LIN {X 0,Y 234.996,Z 198.211,A -85,B 0,C 180,E1 -19773.794,E2 -19773.794} C_VEL
LIN {X 0,Y 235.014,Z 198.209,A -85,B 0,C 180,E1 -19778.97,E2 -19778.97} C_VEL
LIN {X 0,Y 235.098,Z 198.197,A -85,B 0,C 180,E1 -19783.059,E2 -19783.059} C_VEL
LIN {X 0,Y 235.115,Z 198.198,A -85,B 0,C 180,E1 -19787.922,E2 -19787.922} C_VEL
LIN {X 0,Y 235.32,Z 198.173,A -85,B 0,C 180,E1 -19791.412,E2 -19791.412} C_VEL
LIN {X 0,Y 235.356,Z 198.167,A -85,B 0,C 180,E1 -19793.14,E2 -19793.14} C_VEL
LIN {X 0,Y 235.595,Z 198.137,A -85,B 0,C 180,E1 -19798.29,E2 -19798.29} C_VEL
LIN {X 0,Y 235.595,Z 198.138,A -85,B 0,C 180,E1 -19801.709,E2 -19801.709} C_VEL
LIN {X 0,Y 235.351,Z 198.171,A -85,B 0,C 180,E1 -19806.86,E2 -19806.86} C_VEL
LIN {X 0,Y 235.216,Z 198.186,A -85,B 0,C 180,E1 -19810.327,E2 -19810.327} C_VEL
LIN {X 0,Y 235.116,Z 198.199,A -85,B 0,C 180,E1 -19815.606,E2 -19815.606} C_VEL
LIN {X 0,Y 235.009,Z 198.212,A -85,B 0,C 180,E1 -19819.206,E2 -19819.206} C_VEL
LIN {X 0,Y 234.954,Z 198.218,A -85,B 0,C 180,E1 -19822.884,E2 -19822.884} C_VEL
LIN {X 0,Y 234.969,Z 198.217,A -85,B 0,C 180,E1 -19826.657,E2 -19826.657} C_VEL
LIN {X 0,Y 234.924,Z 198.224,A -85,B 0,C 180,E1 -19830.569,E2 -19830.569} C_VEL
LIN {X 0,Y 234.927,Z 198.224,A -85,B 0,C 180,E1 -19834.639,E2 -19834.639} C_VEL
LIN {X 0,Y 234.931,Z 198.302,A -85,B 0,C 180,E1 -19837.285,E2 -19837.285} C_VEL
LIN {X 0,Y 235.419,Z 201.2,A -85,B 0,C 180,E1 -19841.054,E2 -19841.054} C_VEL
LIN {X 0,Y 236.071,Z 204.999,A -85,B 0,C 180,E1 -19845.602,E2 -19845.602} C_VEL
LIN {X 0,Y 236.628,Z 208.216,A -85,B 0,C 180,E1 -19849.2,E2 -19849.2} C_VEL
LIN {X 0,Y 236.793,Z 209.756,A -85,B 0,C 180,E1 -19850.844,E2 -19850.844} C_VEL
LIN {X 0,Y 236.138,Z 210.744,A -85,B 0,C 180,E1 -19851.757,E2 -19851.757} C_VEL
LIN {X 0,Y 233.277,Z 212.555,A -85,B 0,C 180,E1 -19853.17,E2 -19853.17} C_VEL
LIN {X 0,Y 230.314,Z 214.382,A -85,B 0,C 180,E1 -19854.615,E2 -19854.615} C_VEL
LIN {X 0,Y 229.548,Z 215.411,A -85,B 0,C 180,E1 -19855.565,E2 -19855.565} C_VEL
LIN {X 0,Y 229.157,Z 217.081,A -85,B 0,C 180,E1 -19857.204,E2 -19857.204} C_VEL
LIN {X 0,Y 230.079,Z 220.478,A -85,B 0,C 180,E1 -19857.555,E2 -19857.555} C_VEL
LIN {X 0,Y 233.635,Z 233.062,A -85,B 0,C 180,E1 -19858.962,E2 -19858.962} C_VEL
LIN {X 0,Y 236.089,Z 245.694,A -85,B 0,C 180,E1 -19860.544,E2 -19860.544} C_VEL
LIN {X 0,Y 237.459,Z 257.416,A -85,B 0,C 180,E1 -19862.24,E2 -19862.24} C_VEL
LIN {X 0,Y 237.895,Z 268.917,A -85,B 0,C 180,E1 -19864.167,E2 -19864.167} C_VEL
LIN {X 0,Y 237.714,Z 273.85,A -85,B 0,C 180,E1 -19865.083,E2 -19865.083} C_VEL
LIN {X 0,Y 235.107,Z 284.313,A -85,B 0,C 180,E1 -19867.132,E2 -19867.132} C_VEL
LIN {X 0,Y 232.903,Z 293.005,A -85,B 0,C 180,E1 -19869.3,E2 -19869.3} C_VEL
LIN {X 0,Y 230.721,Z 301.061,A -85,B 0,C 180,E1 -19871.806,E2 -19871.806} C_VEL
LIN {X 0,Y 228.899,Z 307.733,A -85,B 0,C 180,E1 -19874.415,E2 -19874.415} C_VEL
LIN {X 0,Y 227.307,Z 313.84,A -85,B 0,C 180,E1 -19877.5,E2 -19877.5} C_VEL
LIN {X 0,Y 226.433,Z 317.814,A -85,B 0,C 180,E1 -19880.171,E2 -19880.171} C_VEL
LIN {X 0,Y 225.852,Z 320.751,A -85,B 0,C 180,E1 -19882.849,E2 -19882.849} C_VEL
LIN {X 0,Y 225.617,Z 322.647,A -85,B 0,C 180,E1 -19885.419,E2 -19885.419} C_VEL
LIN {X 0,Y 225.662,Z 323.764,A -85,B 0,C 180,E1 -19888.215,E2 -19888.215} C_VEL
LIN {X 0,Y 225.698,Z 323.979,A -85,B 0,C 180,E1 -19890,E2 -19890} C_VEL
LIN {X 0,Y 225.662,Z 323.756,A -85,B 0,C 180,E1 -19891.784,E2 -19891.784} C_VEL
LIN {X 0,Y 225.69,Z 322.134,A -85,B 0,C 180,E1 -19895.36,E2 -19895.36} C_VEL
LIN {X 0,Y 225.852,Z 320.726,A -85,B 0,C 180,E1 -19897.15,E2 -19897.15} C_VEL
LIN {X 0,Y 226.432,Z 317.777,A -85,B 0,C 180,E1 -19899.829,E2 -19899.829} C_VEL
LIN {X 0,Y 227.306,Z 313.787,A -85,B 0,C 180,E1 -19902.499,E2 -19902.499} C_VEL
LIN {X 0,Y 228.896,Z 307.66,A -85,B 0,C 180,E1 -19905.584,E2 -19905.584} C_VEL
LIN {X 0,Y 230.72,Z 300.972,A -85,B 0,C 180,E1 -19908.193,E2 -19908.193} C_VEL
LIN {X 0,Y 232.846,Z 293.03,A -85,B 0,C 180,E1 -19910.662,E2 -19910.662} C_VEL
LIN {X 0,Y 235.071,Z 284.172,A -85,B 0,C 180,E1 -19912.871,E2 -19912.871} C_VEL
LIN {X 0,Y 237.68,Z 273.673,A -85,B 0,C 180,E1 -19914.92,E2 -19914.92} C_VEL
LIN {X 0,Y 237.822,Z 264.985,A -85,B 0,C 180,E1 -19916.493,E2 -19916.493} C_VEL
LIN {X 0,Y 237.081,Z 253.496,A -85,B 0,C 180,E1 -19918.313,E2 -19918.313} C_VEL
LIN {X 0,Y 235.519,Z 242.287,A -85,B 0,C 180,E1 -19919.86,E2 -19919.86} C_VEL
LIN {X 0,Y 232.684,Z 229.401,A -85,B 0,C 180,E1 -19921.431,E2 -19921.431} C_VEL
LIN {X 0,Y 229.162,Z 217.507,A -85,B 0,C 180,E1 -19922.7,E2 -19922.7} C_VEL
LIN {X 0,Y 229.124,Z 217.065,A -85,B 0,C 180,E1 -19922.774,E2 -19922.774} C_VEL
LIN {X 0,Y 229.714,Z 214.269,A -85,B 0,C 180,E1 -19925.541,E2 -19925.541} C_VEL
LIN {X 0,Y 229.838,Z 211.122,A -85,B 0,C 180,E1 -19928.817,E2 -19928.817} C_VEL
LIN {X 0,Y 229.356,Z 207.677,A -85,B 0,C 180,E1 -19932.658,E2 -19932.658} C_VEL
LIN {X 0,Y 228.641,Z 203.611,A -85,B 0,C 180,E1 -19937.536,E2 -19937.536} C_VEL
LIN {X 0,Y 228.102,Z 200.24,A -85,B 0,C 180,E1 -19941.96,E2 -19941.96} C_VEL
LIN {X 0,Y 227.872,Z 199.103,A -85,B 0,C 180,E1 -19943.708,E2 -19943.708} C_VEL
LIN {X 0,Y 227.865,Z 199.102,A -85,B 0,C 180,E1 -19948.377,E2 -19948.377} C_VEL
LIN {X 0,Y 227.877,Z 199.101,A -85,B 0,C 180,E1 -19952.444,E2 -19952.444} C_VEL
LIN {X 0,Y 227.905,Z 199.099,A -85,B 0,C 180,E1 -19956.366,E2 -19956.366} C_VEL
LIN {X 0,Y 227.936,Z 199.094,A -85,B 0,C 180,E1 -19960.174,E2 -19960.174} C_VEL
LIN {X 0,Y 228.056,Z 199.078,A -85,B 0,C 180,E1 -19963.898,E2 -19963.898} C_VEL
LIN {X 0,Y 228.07,Z 199.075,A -85,B 0,C 180,E1 -19967.543,E2 -19967.543} C_VEL
LIN {X 0,Y 228.251,Z 199.053,A -85,B 0,C 180,E1 -19971.144,E2 -19971.144} C_VEL
LIN {X 0,Y 228.3,Z 199.047,A -85,B 0,C 180,E1 -19972.927,E2 -19972.927} C_VEL
LIN {X 0,Y 228.55,Z 199.014,A -85,B 0,C 180,E1 -19978.238,E2 -19978.238} C_VEL
LIN {X 0,Y 228.55,Z 199.014,A -85,B 0,C 180,E1 -19981.762,E2 -19981.762} C_VEL
LIN {X 0,Y 228.305,Z 199.045,A -85,B 0,C 180,E1 -19987.073,E2 -19987.073} C_VEL
LIN {X 0,Y 228.144,Z 199.067,A -85,B 0,C 180,E1 -19990.651,E2 -19990.651} C_VEL
LIN {X 0,Y 228.063,Z 199.078,A -85,B 0,C 180,E1 -19994.272,E2 -19994.272} C_VEL
LIN {X 0,Y 228.002,Z 199.084,A -85,B 0,C 180,E1 -19997.954,E2 -19997.954} C_VEL
LIN {X 0,Y 227.929,Z 199.093,A -85,B 0,C 180,E1 -20002.33,E2 -20002.33} C_VEL
LIN {X 0,Y 227.942,Z 199.091,A -85,B 0,C 180,E1 -20006.603,E2 -20006.603} C_VEL
LIN {X 0,Y 227.907,Z 199.096,A -85,B 0,C 180,E1 -20010.296,E2 -20010.296} C_VEL
LIN {X 0,Y 227.875,Z 199.102,A -85,B 0,C 180,E1 -20013.721,E2 -20013.721} C_VEL
LIN {X 0,Y 227.839,Z 199.106,A -85,B 0,C 180,E1 -20018.092,E2 -20018.092} C_VEL
LIN {X 0,Y 227.805,Z 199.11,A -85,B 0,C 180,E1 -20022.744,E2 -20022.744} C_VEL
LIN {X 0,Y 227.825,Z 199.107,A -85,B 0,C 180,E1 -20025.195,E2 -20025.195} C_VEL
LIN {X 0,Y 227.904,Z 199.685,A -85,B 0,C 180,E1 -20027.74,E2 -20027.74} C_VEL
LIN {X 0,Y 228.203,Z 202.454,A -85,B 0,C 180,E1 -20031.98,E2 -20031.98} C_VEL
LIN {X 0,Y 228.228,Z 204.017,A -85,B 0,C 180,E1 -20034.192,E2 -20034.192} C_VEL
LIN {X 0,Y 228.051,Z 206.435,A -85,B 0,C 180,E1 -20037.19,E2 -20037.19} C_VEL
LIN {X 0,Y 229.183,Z 209.556,A -85,B 0,C 180,E1 -20037.548,E2 -20037.548} C_VEL
LIN {X 0,Y 233.35,Z 220.919,A -85,B 0,C 180,E1 -20039.001,E2 -20039.001} C_VEL
LIN {X 0,Y 236.465,Z 231.896,A -85,B 0,C 180,E1 -20040.528,E2 -20040.528} C_VEL
LIN {X 0,Y 238.564,Z 242.208,A -85,B 0,C 180,E1 -20042.103,E2 -20042.103} C_VEL
LIN {X 0,Y 239.656,Z 251.285,A -85,B 0,C 180,E1 -20043.631,E2 -20043.631} C_VEL
LIN {X 0,Y 239.798,Z 255.538,A -85,B 0,C 180,E1 -20044.387,E2 -20044.387} C_VEL
LIN {X 0,Y 237.438,Z 265.983,A -85,B 0,C 180,E1 -20046.217,E2 -20046.217} C_VEL
LIN {X 0,Y 235.445,Z 274.952,A -85,B 0,C 180,E1 -20048.209,E2 -20048.209} C_VEL
LIN {X 0,Y 233.002,Z 283.746,A -85,B 0,C 180,E1 -20050.623,E2 -20050.623} C_VEL
LIN {X 0,Y 230.82,Z 291.15,A -85,B 0,C 180,E1 -20053.187,E2 -20053.187} C_VEL
LIN {X 0,Y 229.103,Z 297.087,A -85,B 0,C 180,E1 -20055.794,E2 -20055.794} C_VEL
LIN {X 0,Y 227.751,Z 301.777,A -85,B 0,C 180,E1 -20058.43,E2 -20058.43} C_VEL
LIN {X 0,Y 226.85,Z 305.362,A -85,B 0,C 180,E1 -20061.089,E2 -20061.089} C_VEL
LIN {X 0,Y 226.238,Z 307.944,A -85,B 0,C 180,E1 -20063.759,E2 -20063.759} C_VEL
LIN {X 0,Y 225.888,Z 309.593,A -85,B 0,C 180,E1 -20066.433,E2 -20066.433} C_VEL
LIN {X 0,Y 225.781,Z 310.2,A -85,B 0,C 180,E1 -20068.217,E2 -20068.217} C_VEL
LIN {X 0,Y 225.751,Z 310.428,A -85,B 0,C 180,E1 -20070,E2 -20070} C_VEL
LIN {X 0,Y 225.781,Z 310.234,A -85,B 0,C 180,E1 -20071.784,E2 -20071.784} C_VEL
LIN {X 0,Y 225.886,Z 309.648,A -85,B 0,C 180,E1 -20073.568,E2 -20073.568} C_VEL
LIN {X 0,Y 226.395,Z 307.325,A -85,B 0,C 180,E1 -20077.133,E2 -20077.133} C_VEL
LIN {X 0,Y 227.097,Z 304.458,A -85,B 0,C 180,E1 -20079.8,E2 -20079.8} C_VEL
LIN {X 0,Y 228.133,Z 300.57,A -85,B 0,C 180,E1 -20082.454,E2 -20082.454} C_VEL
LIN {X 0,Y 229.598,Z 295.549,A -85,B 0,C 180,E1 -20085.081,E2 -20085.081} C_VEL
LIN {X 0,Y 231.424,Z 289.226,A -85,B 0,C 180,E1 -20087.679,E2 -20087.679} C_VEL
LIN {X 0,Y 233.778,Z 281.307,A -85,B 0,C 180,E1 -20090.226,E2 -20090.226} C_VEL
LIN {X 0,Y 235.841,Z 273.317,A -85,B 0,C 180,E1 -20092.311,E2 -20092.311} C_VEL
LIN {X 0,Y 238.119,Z 263.394,A -85,B 0,C 180,E1 -20094.407,E2 -20094.407} C_VEL
LIN {X 0,Y 239.946,Z 254.985,A -85,B 0,C 180,E1 -20095.829,E2 -20095.829} C_VEL
LIN {X 0,Y 239.038,Z 245.57,A -85,B 0,C 180,E1 -20097.485,E2 -20097.485} C_VEL
LIN {X 0,Y 237.134,Z 234.687,A -85,B 0,C 180,E1 -20099.199,E2 -20099.199} C_VEL
LIN {X 0,Y 234.237,Z 223.714,A -85,B 0,C 180,E1 -20100.768,E2 -20100.768} C_VEL
LIN {X 0,Y 230.381,Z 212.541,A -85,B 0,C 180,E1 -20102.23,E2 -20102.23} C_VEL
LIN {X 0,Y 228.147,Z 206.8,A -85,B 0,C 180,E1 -20102.921,E2 -20102.921} C_VEL
LIN {X 0,Y 228.042,Z 206.204,A -85,B 0,C 180,E1 -20103.008,E2 -20103.008} C_VEL
LIN {X 0,Y 228.249,Z 203.403,A -85,B 0,C 180,E1 -20106.816,E2 -20106.816} C_VEL
LIN {X 0,Y 228.079,Z 201.029,A -85,B 0,C 180,E1 -20110.323,E2 -20110.323} C_VEL
LIN {X 0,Y 227.866,Z 199.496,A -85,B 0,C 180,E1 -20112.73,E2 -20112.73} C_VEL
LIN {X 0,Y 227.824,Z 199.105,A -85,B 0,C 180,E1 -20115.196,E2 -20115.196} C_VEL
LIN {X 0,Y 227.827,Z 199.107,A -85,B 0,C 180,E1 -20119.623,E2 -20119.623} C_VEL
LIN {X 0,Y 227.867,Z 199.102,A -85,B 0,C 180,E1 -20124.125,E2 -20124.125} C_VEL
LIN {X 0,Y 227.868,Z 199.1,A -85,B 0,C 180,E1 -20128.377,E2 -20128.377} C_VEL
LIN {X 0,Y 227.881,Z 199.1,A -85,B 0,C 180,E1 -20132.444,E2 -20132.444} C_VEL
LIN {X 0,Y 227.916,Z 199.095,A -85,B 0,C 180,E1 -20136.367,E2 -20136.367} C_VEL
LIN {X 0,Y 227.945,Z 199.092,A -85,B 0,C 180,E1 -20140.175,E2 -20140.175} C_VEL
LIN {X 0,Y 228.06,Z 199.078,A -85,B 0,C 180,E1 -20143.898,E2 -20143.898} C_VEL
LIN {X 0,Y 228.074,Z 199.076,A -85,B 0,C 180,E1 -20147.543,E2 -20147.543} C_VEL
LIN {X 0,Y 228.259,Z 199.051,A -85,B 0,C 180,E1 -20151.144,E2 -20151.144} C_VEL
LIN {X 0,Y 228.308,Z 199.045,A -85,B 0,C 180,E1 -20152.927,E2 -20152.927} C_VEL
LIN {X 0,Y 228.553,Z 199.014,A -85,B 0,C 180,E1 -20158.238,E2 -20158.238} C_VEL
LIN {X 0,Y 228.554,Z 199.015,A -85,B 0,C 180,E1 -20161.762,E2 -20161.762} C_VEL
LIN {X 0,Y 228.303,Z 199.048,A -85,B 0,C 180,E1 -20167.073,E2 -20167.073} C_VEL
LIN {X 0,Y 228.148,Z 199.069,A -85,B 0,C 180,E1 -20170.651,E2 -20170.651} C_VEL
LIN {X 0,Y 228.067,Z 199.078,A -85,B 0,C 180,E1 -20174.272,E2 -20174.272} C_VEL
LIN {X 0,Y 228.005,Z 199.086,A -85,B 0,C 180,E1 -20177.953,E2 -20177.953} C_VEL
LIN {X 0,Y 227.918,Z 199.095,A -85,B 0,C 180,E1 -20182.321,E2 -20182.321} C_VEL
LIN {X 0,Y 227.943,Z 199.093,A -85,B 0,C 180,E1 -20186.602,E2 -20186.602} C_VEL
LIN {X 0,Y 227.898,Z 199.1,A -85,B 0,C 180,E1 -20190.291,E2 -20190.291} C_VEL
LIN {X 0,Y 227.878,Z 199.104,A -85,B 0,C 180,E1 -20193.72,E2 -20193.72} C_VEL
LIN {X 0,Y 227.898,Z 199.226,A -85,B 0,C 180,E1 -20196.536,E2 -20196.536} C_VEL
LIN {X 0,Y 228.347,Z 201.962,A -85,B 0,C 180,E1 -20200.266,E2 -20200.266} C_VEL
LIN {X 0,Y 228.97,Z 205.655,A -85,B 0,C 180,E1 -20204.907,E2 -20204.907} C_VEL
LIN {X 0,Y 229.573,Z 209.041,A -85,B 0,C 180,E1 -20208.839,E2 -20208.839} C_VEL
LIN {X 0,Y 229.805,Z 212.223,A -85,B 0,C 180,E1 -20212.291,E2 -20212.291} C_VEL
LIN {X 0,Y 229.548,Z 215.411,A -85,B 0,C 180,E1 -20215.565,E2 -20215.565} C_VEL
LIN {X 0,Y 229.593,Z 217.095,A -85,B 0,C 180,E1 -20216.397,E2 -20216.397} C_VEL
LIN {X 0,Y 229.787,Z 219.822,A -85,B 0,C 180,E1 -20217.055,E2 -20217.055} C_VEL
LIN {X 0,Y 229.991,Z 225.007,A -85,B 0,C 180,E1 -20217.764,E2 -20217.764} C_VEL
LIN {X 0,Y 229.616,Z 235.258,A -85,B 0,C 180,E1 -20218.556,E2 -20218.556} C_VEL
LIN {X 0,Y 228.975,Z 241.389,A -85,B 0,C 180,E1 -20219.076,E2 -20219.076} C_VEL
LIN {X 0,Y 229.077,Z 243.326,A -85,B 0,C 180,E1 -20219.308,E2 -20219.308} C_VEL
LIN {X 0,Y 230.659,Z 255.124,A -85,B 0,C 180,E1 -20221.043,E2 -20221.043} C_VEL
LIN {X 0,Y 231.247,Z 266.076,A -85,B 0,C 180,E1 -20222.878,E2 -20222.878} C_VEL
LIN {X 0,Y 231.01,Z 274.817,A -85,B 0,C 180,E1 -20224.55,E2 -20224.55} C_VEL
LIN {X 0,Y 228.563,Z 284.102,A -85,B 0,C 180,E1 -20226.438,E2 -20226.438} C_VEL
LIN {X 0,Y 226.032,Z 293.522,A -85,B 0,C 180,E1 -20228.874,E2 -20228.874} C_VEL
LIN {X 0,Y 223.962,Z 300.849,A -85,B 0,C 180,E1 -20231.237,E2 -20231.237} C_VEL
LIN {X 0,Y 222.046,Z 307.521,A -85,B 0,C 180,E1 -20233.922,E2 -20233.922} C_VEL
LIN {X 0,Y 220.351,Z 313.627,A -85,B 0,C 180,E1 -20237.099,E2 -20237.099} C_VEL
LIN {X 0,Y 219.405,Z 317.601,A -85,B 0,C 180,E1 -20239.852,E2 -20239.852} C_VEL
LIN {X 0,Y 218.803,Z 320.538,A -85,B 0,C 180,E1 -20242.618,E2 -20242.618} C_VEL
LIN {X 0,Y 218.52,Z 322.61,A -85,B 0,C 180,E1 -20245.574,E2 -20245.574} C_VEL
LIN {X 0,Y 218.56,Z 323.551,A -85,B 0,C 180,E1 -20248.157,E2 -20248.157} C_VEL
LIN {X 0,Y 218.614,Z 323.766,A -85,B 0,C 180,E1 -20250,E2 -20250} C_VEL
LIN {X 0,Y 218.56,Z 323.542,A -85,B 0,C 180,E1 -20251.842,E2 -20251.842} C_VEL
LIN {X 0,Y 218.554,Z 322.534,A -85,B 0,C 180,E1 -20254.538,E2 -20254.538} C_VEL
LIN {X 0,Y 218.803,Z 320.512,A -85,B 0,C 180,E1 -20257.381,E2 -20257.381} C_VEL
LIN {X 0,Y 219.404,Z 317.562,A -85,B 0,C 180,E1 -20260.147,E2 -20260.147} C_VEL
LIN {X 0,Y 220.35,Z 313.572,A -85,B 0,C 180,E1 -20262.9,E2 -20262.9} C_VEL
LIN {X 0,Y 222.044,Z 307.444,A -85,B 0,C 180,E1 -20266.078,E2 -20266.078} C_VEL
LIN {X 0,Y 223.96,Z 300.756,A -85,B 0,C 180,E1 -20268.762,E2 -20268.762} C_VEL
LIN {X 0,Y 225.999,Z 293.482,A -85,B 0,C 180,E1 -20271.104,E2 -20271.104} C_VEL
LIN {X 0,Y 228.517,Z 283.955,A -85,B 0,C 180,E1 -20273.566,E2 -20273.566} C_VEL
LIN {X 0,Y 231.127,Z 273.451,A -85,B 0,C 180,E1 -20275.677,E2 -20275.677} C_VEL
LIN {X 0,Y 231.116,Z 262.504,A -85,B 0,C 180,E1 -20277.709,E2 -20277.709} C_VEL
LIN {X 0,Y 230.318,Z 251.884,A -85,B 0,C 180,E1 -20279.417,E2 -20279.417} C_VEL
LIN {X 0,Y 228.386,Z 239.706,A -85,B 0,C 180,E1 -20281.145,E2 -20281.145} C_VEL
LIN {X 0,Y 225.462,Z 227.374,A -85,B 0,C 180,E1 -20282.687,E2 -20282.687} C_VEL
LIN {X 0,Y 222.418,Z 217.479,A -85,B 0,C 180,E1 -20283.812,E2 -20283.812} C_VEL
LIN {X 0,Y 222.355,Z 216.881,A -85,B 0,C 180,E1 -20283.862,E2 -20283.862} C_VEL
LIN {X 0,Y 222.793,Z 213,A -85,B 0,C 180,E1 -20287.943,E2 -20287.943} C_VEL
LIN {X 0,Y 222.632,Z 210.496,A -85,B 0,C 180,E1 -20290.744,E2 -20290.744} C_VEL
LIN {X 0,Y 222.122,Z 207.666,A -85,B 0,C 180,E1 -20294.113,E2 -20294.113} C_VEL
LIN {X 0,Y 221.554,Z 204.406,A -85,B 0,C 180,E1 -20298.229,E2 -20298.229} C_VEL
LIN {X 0,Y 221.028,Z 201.065,A -85,B 0,C 180,E1 -20302.833,E2 -20302.833} C_VEL
LIN {X 0,Y 220.812,Z 199.981,A -85,B 0,C 180,E1 -20304.489,E2 -20304.489} C_VEL
LIN {X 0,Y 220.832,Z 199.977,A -85,B 0,C 180,E1 -20309.389,E2 -20309.389} C_VEL
LIN {X 0,Y 220.892,Z 199.972,A -85,B 0,C 180,E1 -20313.549,E2 -20313.549} C_VEL
LIN {X 0,Y 220.864,Z 199.976,A -85,B 0,C 180,E1 -20317.552,E2 -20317.552} C_VEL
LIN {X 0,Y 220.983,Z 199.959,A -85,B 0,C 180,E1 -20322.571,E2 -20322.571} C_VEL
LIN {X 0,Y 221.01,Z 199.956,A -85,B 0,C 180,E1 -20327.138,E2 -20327.138} C_VEL
LIN {X 0,Y 221.192,Z 199.931,A -85,B 0,C 180,E1 -20330.859,E2 -20330.859} C_VEL
LIN {X 0,Y 221.122,Z 199.941,A -85,B 0,C 180,E1 -20334.529,E2 -20334.529} C_VEL
LIN {X 0,Y 221.508,Z 199.891,A -85,B 0,C 180,E1 -20338.182,E2 -20338.182} C_VEL
LIN {X 0,Y 221.508,Z 199.891,A -85,B 0,C 180,E1 -20341.818,E2 -20341.818} C_VEL
LIN {X 0,Y 221.243,Z 199.924,A -85,B 0,C 180,E1 -20347.3,E2 -20347.3} C_VEL
LIN {X 0,Y 221.066,Z 199.948,A -85,B 0,C 180,E1 -20350.997,E2 -20350.997} C_VEL
LIN {X 0,Y 220.994,Z 199.956,A -85,B 0,C 180,E1 -20354.739,E2 -20354.739} C_VEL
LIN {X 0,Y 220.921,Z 199.966,A -85,B 0,C 180,E1 -20358.55,E2 -20358.55} C_VEL
LIN {X 0,Y 220.895,Z 199.968,A -85,B 0,C 180,E1 -20362.683,E2 -20362.683} C_VEL
LIN {X 0,Y 220.885,Z 199.971,A -85,B 0,C 180,E1 -20367.016,E2 -20367.016} C_VEL
LIN {X 0,Y 220.837,Z 199.976,A -85,B 0,C 180,E1 -20370.768,E2 -20370.768} C_VEL
LIN {X 0,Y 220.792,Z 199.983,A -85,B 0,C 180,E1 -20374.957,E2 -20374.957} C_VEL
LIN {X 0,Y 220.8,Z 199.98,A -85,B 0,C 180,E1 -20377.276,E2 -20377.276} C_VEL
LIN {X 0,Y 220.794,Z 199.982,A -85,B 0,C 180,E1 -20380.189,E2 -20380.189} C_VEL
LIN {X 0,Y 220.767,Z 199.986,A -85,B 0,C 180,E1 -20384.456,E2 -20384.456} C_VEL
LIN {X 0,Y 220.776,Z 199.984,A -85,B 0,C 180,E1 -20385.547,E2 -20385.547} C_VEL
LIN {X 0,Y 220.949,Z 201.161,A -85,B 0,C 180,E1 -20388.09,E2 -20388.09} C_VEL
LIN {X 0,Y 221.149,Z 202.697,A -85,B 0,C 180,E1 -20390.537,E2 -20390.537} C_VEL
LIN {X 0,Y 221.222,Z 204.251,A -85,B 0,C 180,E1 -20392.872,E2 -20392.872} C_VEL
LIN {X 0,Y 221.073,Z 206.476,A -85,B 0,C 180,E1 -20396.005,E2 -20396.005} C_VEL
LIN {X 0,Y 222.205,Z 209.663,A -85,B 0,C 180,E1 -20396.386,E2 -20396.386} C_VEL
LIN {X 0,Y 226.427,Z 220.676,A -85,B 0,C 180,E1 -20397.899,E2 -20397.899} C_VEL
LIN {X 0,Y 229.58,Z 231.463,A -85,B 0,C 180,E1 -20399.474,E2 -20399.474} C_VEL
LIN {X 0,Y 231.954,Z 242.834,A -85,B 0,C 180,E1 -20401.291,E2 -20401.291} C_VEL
LIN {X 0,Y 233.148,Z 253.158,A -85,B 0,C 180,E1 -20403.118,E2 -20403.118} C_VEL
LIN {X 0,Y 233.139,Z 257.042,A -85,B 0,C 180,E1 -20403.841,E2 -20403.841} C_VEL
LIN {X 0,Y 230.721,Z 267.252,A -85,B 0,C 180,E1 -20405.719,E2 -20405.719} C_VEL
LIN {X 0,Y 228.477,Z 276.713,A -85,B 0,C 180,E1 -20407.955,E2 -20407.955} C_VEL
LIN {X 0,Y 225.927,Z 285.309,A -85,B 0,C 180,E1 -20410.464,E2 -20410.464} C_VEL
LIN {X 0,Y 223.73,Z 292.473,A -85,B 0,C 180,E1 -20413.109,E2 -20413.109} C_VEL
LIN {X 0,Y 222.221,Z 297.302,A -85,B 0,C 180,E1 -20415.345,E2 -20415.345} C_VEL
LIN {X 0,Y 220.806,Z 301.992,A -85,B 0,C 180,E1 -20418.06,E2 -20418.06} C_VEL
LIN {X 0,Y 219.831,Z 305.576,A -85,B 0,C 180,E1 -20420.802,E2 -20420.802} C_VEL
LIN {X 0,Y 219.119,Z 308.408,A -85,B 0,C 180,E1 -20423.878,E2 -20423.878} C_VEL
LIN {X 0,Y 218.8,Z 309.806,A -85,B 0,C 180,E1 -20426.317,E2 -20426.317} C_VEL
LIN {X 0,Y 218.7,Z 310.413,A -85,B 0,C 180,E1 -20428.159,E2 -20428.159} C_VEL
LIN {X 0,Y 218.666,Z 310.641,A -85,B 0,C 180,E1 -20430,E2 -20430} C_VEL
LIN {X 0,Y 218.699,Z 310.447,A -85,B 0,C 180,E1 -20431.842,E2 -20431.842} C_VEL
LIN {X 0,Y 219.015,Z 308.894,A -85,B 0,C 180,E1 -20435.525,E2 -20435.525} C_VEL
LIN {X 0,Y 219.352,Z 307.537,A -85,B 0,C 180,E1 -20437.364,E2 -20437.364} C_VEL
LIN {X 0,Y 220.097,Z 304.671,A -85,B 0,C 180,E1 -20440.115,E2 -20440.115} C_VEL
LIN {X 0,Y 221.208,Z 300.781,A -85,B 0,C 180,E1 -20442.85,E2 -20442.85} C_VEL
LIN {X 0,Y 222.754,Z 295.761,A -85,B 0,C 180,E1 -20445.556,E2 -20445.556} C_VEL
LIN {X 0,Y 224.669,Z 289.437,A -85,B 0,C 180,E1 -20448.229,E2 -20448.229} C_VEL
LIN {X 0,Y 227.143,Z 281.517,A -85,B 0,C 180,E1 -20450.844,E2 -20450.844} C_VEL
LIN {X 0,Y 229.155,Z 274.045,A -85,B 0,C 180,E1 -20452.859,E2 -20452.859} C_VEL
LIN {X 0,Y 231.392,Z 264.669,A -85,B 0,C 180,E1 -20454.925,E2 -20454.925} C_VEL
LIN {X 0,Y 233.283,Z 256.481,A -85,B 0,C 180,E1 -20456.383,E2 -20456.383} C_VEL
LIN {X 0,Y 232.765,Z 248.766,A -85,B 0,C 180,E1 -20457.823,E2 -20457.823} C_VEL
LIN {X 0,Y 231.143,Z 238.24,A -85,B 0,C 180,E1 -20459.606,E2 -20459.606} C_VEL
LIN {X 0,Y 228.364,Z 226.928,A -85,B 0,C 180,E1 -20461.348,E2 -20461.348} C_VEL
LIN {X 0,Y 224.773,Z 216.012,A -85,B 0,C 180,E1 -20462.897,E2 -20462.897} C_VEL
LIN {X 0,Y 221.715,Z 208.654,A -85,B 0,C 180,E1 -20463.908,E2 -20463.908} C_VEL
LIN {X 0,Y 221.098,Z 206.433,A -85,B 0,C 180,E1 -20464.2,E2 -20464.2} C_VEL
LIN {X 0,Y 221.223,Z 204.162,A -85,B 0,C 180,E1 -20467.418,E2 -20467.418} C_VEL
LIN {X 0,Y 221.105,Z 202.278,A -85,B 0,C 180,E1 -20470.283,E2 -20470.283} C_VEL
LIN {X 0,Y 220.87,Z 200.63,A -85,B 0,C 180,E1 -20472.958,E2 -20472.958} C_VEL
LIN {X 0,Y 220.773,Z 199.982,A -85,B 0,C 180,E1 -20474.455,E2 -20474.455} C_VEL
LIN {X 0,Y 220.768,Z 199.985,A -85,B 0,C 180,E1 -20478.047,E2 -20478.047} C_VEL
LIN {X 0,Y 220.808,Z 199.981,A -85,B 0,C 180,E1 -20480.463,E2 -20480.463} C_VEL
LIN {X 0,Y 220.826,Z 199.978,A -85,B 0,C 180,E1 -20482.793,E2 -20482.793} C_VEL
LIN {X 0,Y 220.818,Z 199.977,A -85,B 0,C 180,E1 -20487.244,E2 -20487.244} C_VEL
LIN {X 0,Y 220.829,Z 199.976,A -85,B 0,C 180,E1 -20491.485,E2 -20491.485} C_VEL
LIN {X 0,Y 220.869,Z 199.972,A -85,B 0,C 180,E1 -20495.565,E2 -20495.565} C_VEL
LIN {X 0,Y 220.895,Z 199.969,A -85,B 0,C 180,E1 -20499.514,E2 -20499.514} C_VEL
LIN {X 0,Y 221.019,Z 199.951,A -85,B 0,C 180,E1 -20503.37,E2 -20503.37} C_VEL
LIN {X 0,Y 221.013,Z 199.955,A -85,B 0,C 180,E1 -20507.138,E2 -20507.138} C_VEL
LIN {X 0,Y 221.198,Z 199.93,A -85,B 0,C 180,E1 -20510.859,E2 -20510.859} C_VEL
LIN {X 0,Y 221.125,Z 199.94,A -85,B 0,C 180,E1 -20514.528,E2 -20514.528} C_VEL
LIN {X 0,Y 221.511,Z 199.891,A -85,B 0,C 180,E1 -20518.182,E2 -20518.182} C_VEL
LIN {X 0,Y 221.511,Z 199.892,A -85,B 0,C 180,E1 -20521.818,E2 -20521.818} C_VEL
LIN {X 0,Y 221.241,Z 199.927,A -85,B 0,C 180,E1 -20527.3,E2 -20527.3} C_VEL
LIN {X 0,Y 221.084,Z 199.949,A -85,B 0,C 180,E1 -20530.996,E2 -20530.996} C_VEL
LIN {X 0,Y 221.018,Z 199.956,A -85,B 0,C 180,E1 -20536.63,E2 -20536.63} C_VEL
LIN {X 0,Y 220.886,Z 199.971,A -85,B 0,C 180,E1 -20540.487,E2 -20540.487} C_VEL
LIN {X 0,Y 220.864,Z 199.974,A -85,B 0,C 180,E1 -20544.435,E2 -20544.435} C_VEL
LIN {X 0,Y 220.828,Z 199.98,A -85,B 0,C 180,E1 -20548.515,E2 -20548.515} C_VEL
LIN {X 0,Y 220.818,Z 199.984,A -85,B 0,C 180,E1 -20552.756,E2 -20552.756} C_VEL
LIN {X 0,Y 220.82,Z 199.999,A -85,B 0,C 180,E1 -20555.51,E2 -20555.51} C_VEL
LIN {X 0,Y 221.297,Z 202.725,A -85,B 0,C 180,E1 -20559.432,E2 -20559.432} C_VEL
LIN {X 0,Y 221.873,Z 206.346,A -85,B 0,C 180,E1 -20564.176,E2 -20564.176} C_VEL
LIN {X 0,Y 222.52,Z 209.855,A -85,B 0,C 180,E1 -20568.451,E2 -20568.451} C_VEL
LIN {X 0,Y 222.776,Z 213.061,A -85,B 0,C 180,E1 -20572.063,E2 -20572.063} C_VEL
LIN {X 0,Y 222.394,Z 216.878,A -85,B 0,C 180,E1 -20576.09,E2 -20576.09} C_VEL
LIN {X 0,Y 223.259,Z 220.158,A -85,B 0,C 180,E1 -20576.43,E2 -20576.43} C_VEL
LIN {X 0,Y 226.726,Z 232.025,A -85,B 0,C 180,E1 -20577.837,E2 -20577.837} C_VEL
LIN {X 0,Y 229.077,Z 243.326,A -85,B 0,C 180,E1 -20579.308,E2 -20579.308} C_VEL
LIN {X 0,Y 229.206,Z 248.711,A -85,B 0,C 180,E1 -20579.969,E2 -20579.969} C_VEL
LIN {X 0,Y 227.453,Z 257.649,A -85,B 0,C 180,E1 -20580.995,E2 -20580.995} C_VEL
LIN {X 0,Y 225.218,Z 266.215,A -85,B 0,C 180,E1 -20582.153,E2 -20582.153} C_VEL
LIN {X 0,Y 224.605,Z 270.988,A -85,B 0,C 180,E1 -20583.006,E2 -20583.006} C_VEL
LIN {X 0,Y 224.313,Z 275.736,A -85,B 0,C 180,E1 -20583.983,E2 -20583.983} C_VEL
LIN {X 0,Y 221.528,Z 285.687,A -85,B 0,C 180,E1 -20586.14,E2 -20586.14} C_VEL
LIN {X 0,Y 219.19,Z 294.001,A -85,B 0,C 180,E1 -20588.411,E2 -20588.411} C_VEL
LIN {X 0,Y 216.839,Z 301.874,A -85,B 0,C 180,E1 -20591.088,E2 -20591.088} C_VEL
LIN {X 0,Y 214.907,Z 308.304,A -85,B 0,C 180,E1 -20593.86,E2 -20593.86} C_VEL
LIN {X 0,Y 213.382,Z 313.413,A -85,B 0,C 180,E1 -20596.67,E2 -20596.67} C_VEL
LIN {X 0,Y 212.399,Z 317.388,A -85,B 0,C 180,E1 -20599.514,E2 -20599.514} C_VEL
LIN {X 0,Y 211.734,Z 320.325,A -85,B 0,C 180,E1 -20602.37,E2 -20602.37} C_VEL
LIN {X 0,Y 211.42,Z 322.542,A -85,B 0,C 180,E1 -20605.758,E2 -20605.758} C_VEL
LIN {X 0,Y 211.46,Z 323.338,A -85,B 0,C 180,E1 -20608.095,E2 -20608.095} C_VEL
LIN {X 0,Y 211.531,Z 323.554,A -85,B 0,C 180,E1 -20610,E2 -20610} C_VEL
LIN {X 0,Y 211.46,Z 323.329,A -85,B 0,C 180,E1 -20611.904,E2 -20611.904} C_VEL
LIN {X 0,Y 211.473,Z 322.447,A -85,B 0,C 180,E1 -20614.434,E2 -20614.434} C_VEL
LIN {X 0,Y 211.734,Z 320.298,A -85,B 0,C 180,E1 -20617.629,E2 -20617.629} C_VEL
LIN {X 0,Y 212.398,Z 317.347,A -85,B 0,C 180,E1 -20620.485,E2 -20620.485} C_VEL
LIN {X 0,Y 213.381,Z 313.356,A -85,B 0,C 180,E1 -20623.329,E2 -20623.329} C_VEL
LIN {X 0,Y 215.185,Z 307.228,A -85,B 0,C 180,E1 -20626.605,E2 -20626.605} C_VEL
LIN {X 0,Y 217.235,Z 300.54,A -85,B 0,C 180,E1 -20629.366,E2 -20629.366} C_VEL
LIN {X 0,Y 219.618,Z 292.343,A -85,B 0,C 180,E1 -20632.053,E2 -20632.053} C_VEL
LIN {X 0,Y 222.012,Z 283.738,A -85,B 0,C 180,E1 -20634.3,E2 -20634.3} C_VEL
LIN {X 0,Y 224.468,Z 274.411,A -85,B 0,C 180,E1 -20636.247,E2 -20636.247} C_VEL
LIN {X 0,Y 224.571,Z 263.404,A -85,B 0,C 180,E1 -20638.39,E2 -20638.39} C_VEL
LIN {X 0,Y 223.852,Z 253.028,A -85,B 0,C 180,E1 -20640.154,E2 -20640.154} C_VEL
LIN {X 0,Y 222.016,Z 240.798,A -85,B 0,C 180,E1 -20641.999,E2 -20641.999} C_VEL
LIN {X 0,Y 219.31,Z 229.155,A -85,B 0,C 180,E1 -20643.571,E2 -20643.571} C_VEL
LIN {X 0,Y 215.566,Z 217.029,A -85,B 0,C 180,E1 -20645.049,E2 -20645.049} C_VEL
LIN {X 0,Y 215.524,Z 216.595,A -85,B 0,C 180,E1 -20645.131,E2 -20645.131} C_VEL
LIN {X 0,Y 215.794,Z 213.473,A -85,B 0,C 180,E1 -20648.589,E2 -20648.589} C_VEL
LIN {X 0,Y 215.547,Z 211.076,A -85,B 0,C 180,E1 -20651.416,E2 -20651.416} C_VEL
LIN {X 0,Y 214.866,Z 207.407,A -85,B 0,C 180,E1 -20656.02,E2 -20656.02} C_VEL
LIN {X 0,Y 214.473,Z 205.148,A -85,B 0,C 180,E1 -20659.052,E2 -20659.052} C_VEL
LIN {X 0,Y 213.959,Z 201.888,A -85,B 0,C 180,E1 -20663.754,E2 -20663.754} C_VEL
LIN {X 0,Y 213.767,Z 200.858,A -85,B 0,C 180,E1 -20665.65,E2 -20665.65} C_VEL
LIN {X 0,Y 213.759,Z 200.859,A -85,B 0,C 180,E1 -20670.451,E2 -20670.451} C_VEL
LIN {X 0,Y 213.797,Z 200.856,A -85,B 0,C 180,E1 -20674.701,E2 -20674.701} C_VEL
LIN {X 0,Y 213.802,Z 200.855,A -85,B 0,C 180,E1 -20678.802,E2 -20678.802} C_VEL
LIN {X 0,Y 213.942,Z 200.836,A -85,B 0,C 180,E1 -20682.804,E2 -20682.804} C_VEL
LIN {X 0,Y 213.951,Z 200.834,A -85,B 0,C 180,E1 -20686.706,E2 -20686.706} C_VEL
LIN {X 0,Y 214.132,Z 200.809,A -85,B 0,C 180,E1 -20690.555,E2 -20690.555} C_VEL
LIN {X 0,Y 214.083,Z 200.817,A -85,B 0,C 180,E1 -20694.348,E2 -20694.348} C_VEL
LIN {X 0,Y 214.441,Z 200.771,A -85,B 0,C 180,E1 -20698.122,E2 -20698.122} C_VEL
LIN {X 0,Y 214.549,Z 200.759,A -85,B 0,C 180,E1 -20700,E2 -20700} C_VEL
LIN {X 0,Y 214.44,Z 200.772,A -85,B 0,C 180,E1 -20701.878,E2 -20701.878} C_VEL
LIN {X 0,Y 214.184,Z 200.804,A -85,B 0,C 180,E1 -20707.542,E2 -20707.542} C_VEL
LIN {X 0,Y 213.998,Z 200.828,A -85,B 0,C 180,E1 -20711.365,E2 -20711.365} C_VEL
LIN {X 0,Y 213.932,Z 200.835,A -85,B 0,C 180,E1 -20715.237,E2 -20715.237} C_VEL
LIN {X 0,Y 213.839,Z 200.847,A -85,B 0,C 180,E1 -20719.188,E2 -20719.188} C_VEL
LIN {X 0,Y 213.846,Z 200.847,A -85,B 0,C 180,E1 -20723.227,E2 -20723.227} C_VEL
LIN {X 0,Y 213.828,Z 200.85,A -85,B 0,C 180,E1 -20727.45,E2 -20727.45} C_VEL
LIN {X 0,Y 213.767,Z 200.858,A -85,B 0,C 180,E1 -20731.738,E2 -20731.738} C_VEL
LIN {X 0,Y 213.74,Z 200.861,A -85,B 0,C 180,E1 -20736.289,E2 -20736.289} C_VEL
LIN {X 0,Y 213.71,Z 200.869,A -85,B 0,C 180,E1 -20741.126,E2 -20741.126} C_VEL
LIN {X 0,Y 213.702,Z 200.867,A -85,B 0,C 180,E1 -20743.68,E2 -20743.68} C_VEL
LIN {X 0,Y 213.811,Z 201.421,A -85,B 0,C 180,E1 -20746.349,E2 -20746.349} C_VEL
LIN {X 0,Y 214.054,Z 202.999,A -85,B 0,C 180,E1 -20749.039,E2 -20749.039} C_VEL
LIN {X 0,Y 214.184,Z 204.838,A -85,B 0,C 180,E1 -20751.954,E2 -20751.954} C_VEL
LIN {X 0,Y 214.143,Z 206.819,A -85,B 0,C 180,E1 -20754.748,E2 -20754.748} C_VEL
LIN {X 0,Y 215.271,Z 209.934,A -85,B 0,C 180,E1 -20755.15,E2 -20755.15} C_VEL
LIN {X 0,Y 219.326,Z 219.869,A -85,B 0,C 180,E1 -20756.631,E2 -20756.631} C_VEL
LIN {X 0,Y 222.806,Z 231.303,A -85,B 0,C 180,E1 -20758.394,E2 -20758.394} C_VEL
LIN {X 0,Y 225.13,Z 242.202,A -85,B 0,C 180,E1 -20760.207,E2 -20760.207} C_VEL
LIN {X 0,Y 226.469,Z 252.213,A -85,B 0,C 180,E1 -20762.049,E2 -20762.049} C_VEL
LIN {X 0,Y 226.743,Z 257.261,A -85,B 0,C 180,E1 -20763.044,E2 -20763.044} C_VEL
LIN {X 0,Y 224.259,Z 267.469,A -85,B 0,C 180,E1 -20764.972,E2 -20764.972} C_VEL
LIN {X 0,Y 222.178,Z 275.878,A -85,B 0,C 180,E1 -20766.977,E2 -20766.977} C_VEL
LIN {X 0,Y 219.657,Z 284.177,A -85,B 0,C 180,E1 -20769.394,E2 -20769.394} C_VEL
LIN {X 0,Y 217.259,Z 291.58,A -85,B 0,C 180,E1 -20772.103,E2 -20772.103} C_VEL
LIN {X 0,Y 215.361,Z 297.517,A -85,B 0,C 180,E1 -20774.867,E2 -20774.867} C_VEL
LIN {X 0,Y 213.862,Z 302.206,A -85,B 0,C 180,E1 -20777.667,E2 -20777.667} C_VEL
LIN {X 0,Y 212.837,Z 305.79,A -85,B 0,C 180,E1 -20780.497,E2 -20780.497} C_VEL
LIN {X 0,Y 212.018,Z 308.832,A -85,B 0,C 180,E1 -20783.961,E2 -20783.961} C_VEL
LIN {X 0,Y 211.717,Z 310.019,A -85,B 0,C 180,E1 -20786.194,E2 -20786.194} C_VEL
LIN {X 0,Y 211.62,Z 310.626,A -85,B 0,C 180,E1 -20788.097,E2 -20788.097} C_VEL
LIN {X 0,Y 211.584,Z 310.853,A -85,B 0,C 180,E1 -20790,E2 -20790} C_VEL
LIN {X 0,Y 211.62,Z 310.659,A -85,B 0,C 180,E1 -20791.904,E2 -20791.904} C_VEL
LIN {X 0,Y 211.961,Z 309.106,A -85,B 0,C 180,E1 -20795.709,E2 -20795.709} C_VEL
LIN {X 0,Y 212.307,Z 307.75,A -85,B 0,C 180,E1 -20797.609,E2 -20797.609} C_VEL
LIN {X 0,Y 213.092,Z 304.883,A -85,B 0,C 180,E1 -20800.451,E2 -20800.451} C_VEL
LIN {X 0,Y 214.269,Z 300.994,A -85,B 0,C 180,E1 -20803.274,E2 -20803.274} C_VEL
LIN {X 0,Y 215.926,Z 295.972,A -85,B 0,C 180,E1 -20806.061,E2 -20806.061} C_VEL
LIN {X 0,Y 217.943,Z 289.647,A -85,B 0,C 180,E1 -20808.813,E2 -20808.813} C_VEL
LIN {X 0,Y 220.533,Z 281.727,A -85,B 0,C 180,E1 -20811.499,E2 -20811.499} C_VEL
LIN {X 0,Y 222.948,Z 272.897,A -85,B 0,C 180,E1 -20813.911,E2 -20813.911} C_VEL
LIN {X 0,Y 225.548,Z 262.711,A -85,B 0,C 180,E1 -20816.113,E2 -20816.113} C_VEL
LIN {X 0,Y 226.793,Z 256.695,A -85,B 0,C 180,E1 -20817.199,E2 -20817.199} C_VEL
LIN {X 0,Y 225.714,Z 245.594,A -85,B 0,C 180,E1 -20819.328,E2 -20819.328} C_VEL
LIN {X 0,Y 223.696,Z 234.829,A -85,B 0,C 180,E1 -20821.183,E2 -20821.183} C_VEL
LIN {X 0,Y 220.795,Z 224.168,A -85,B 0,C 180,E1 -20822.868,E2 -20822.868} C_VEL
LIN {X 0,Y 216.615,Z 212.939,A -85,B 0,C 180,E1 -20824.561,E2 -20824.561} C_VEL
LIN {X 0,Y 215.116,Z 209.649,A -85,B 0,C 180,E1 -20825.049,E2 -20825.049} C_VEL
LIN {X 0,Y 214.136,Z 206.649,A -85,B 0,C 180,E1 -20825.49,E2 -20825.49} C_VEL
LIN {X 0,Y 214.164,Z 204.611,A -85,B 0,C 180,E1 -20828.573,E2 -20828.573} C_VEL
LIN {X 0,Y 214.008,Z 203.055,A -85,B 0,C 180,E1 -20831.056,E2 -20831.056} C_VEL
LIN {X 0,Y 213.811,Z 201.501,A -85,B 0,C 180,E1 -20833.685,E2 -20833.685} C_VEL
LIN {X 0,Y 213.704,Z 200.864,A -85,B 0,C 180,E1 -20836.345,E2 -20836.345} C_VEL
LIN {X 0,Y 213.718,Z 200.863,A -85,B 0,C 180,E1 -20839.143,E2 -20839.143} C_VEL
LIN {X 0,Y 213.743,Z 200.861,A -85,B 0,C 180,E1 -20843.711,E2 -20843.711} C_VEL
LIN {X 0,Y 213.782,Z 200.856,A -85,B 0,C 180,E1 -20848.731,E2 -20848.731} C_VEL
LIN {X 0,Y 213.828,Z 200.85,A -85,B 0,C 180,E1 -20852.603,E2 -20852.603} C_VEL
LIN {X 0,Y 213.854,Z 200.844,A -85,B 0,C 180,E1 -20856.953,E2 -20856.953} C_VEL
LIN {X 0,Y 213.946,Z 200.832,A -85,B 0,C 180,E1 -20862.804,E2 -20862.804} C_VEL
LIN {X 0,Y 213.955,Z 200.833,A -85,B 0,C 180,E1 -20866.707,E2 -20866.707} C_VEL
LIN {X 0,Y 214.137,Z 200.809,A -85,B 0,C 180,E1 -20870.555,E2 -20870.555} C_VEL
LIN {X 0,Y 214.087,Z 200.817,A -85,B 0,C 180,E1 -20874.348,E2 -20874.348} C_VEL
LIN {X 0,Y 214.443,Z 200.772,A -85,B 0,C 180,E1 -20878.122,E2 -20878.122} C_VEL
LIN {X 0,Y 214.552,Z 200.757,A -85,B 0,C 180,E1 -20880,E2 -20880} C_VEL
LIN {X 0,Y 214.444,Z 200.773,A -85,B 0,C 180,E1 -20881.878,E2 -20881.878} C_VEL
LIN {X 0,Y 214.183,Z 200.806,A -85,B 0,C 180,E1 -20887.542,E2 -20887.542} C_VEL
LIN {X 0,Y 214.01,Z 200.828,A -85,B 0,C 180,E1 -20891.364,E2 -20891.364} C_VEL
LIN {X 0,Y 213.936,Z 200.838,A -85,B 0,C 180,E1 -20895.237,E2 -20895.237} C_VEL
LIN {X 0,Y 213.838,Z 200.849,A -85,B 0,C 180,E1 -20899.187,E2 -20899.187} C_VEL
LIN {X 0,Y 213.813,Z 200.852,A -85,B 0,C 180,E1 -20903.231,E2 -20903.231} C_VEL
LIN {X 0,Y 213.831,Z 200.85,A -85,B 0,C 180,E1 -20907.45,E2 -20907.45} C_VEL
LIN {X 0,Y 213.769,Z 200.861,A -85,B 0,C 180,E1 -20911.737,E2 -20911.737} C_VEL
LIN {X 0,Y 213.768,Z 200.972,A -85,B 0,C 180,E1 -20914.722,E2 -20914.722} C_VEL
LIN {X 0,Y 214.202,Z 203.513,A -85,B 0,C 180,E1 -20918.564,E2 -20918.564} C_VEL
LIN {X 0,Y 214.803,Z 207.022,A -85,B 0,C 180,E1 -20923.4,E2 -20923.4} C_VEL
LIN {X 0,Y 215.261,Z 209.611,A -85,B 0,C 180,E1 -20926.715,E2 -20926.715} C_VEL
LIN {X 0,Y 215.633,Z 211.738,A -85,B 0,C 180,E1 -20929.318,E2 -20929.318} C_VEL
LIN {X 0,Y 215.722,Z 214.896,A -85,B 0,C 180,E1 -20932.935,E2 -20932.935} C_VEL
LIN {X 0,Y 215.551,Z 216.777,A -85,B 0,C 180,E1 -20934.882,E2 -20934.882} C_VEL
LIN {X 0,Y 216.646,Z 220.245,A -85,B 0,C 180,E1 -20935.28,E2 -20935.28} C_VEL
LIN {X 0,Y 220.386,Z 232.914,A -85,B 0,C 180,E1 -20936.892,E2 -20936.892} C_VEL
LIN {X 0,Y 222.869,Z 245.412,A -85,B 0,C 180,E1 -20938.625,E2 -20938.625} C_VEL
LIN {X 0,Y 224.19,Z 256.508,A -85,B 0,C 180,E1 -20940.365,E2 -20940.365} C_VEL
LIN {X 0,Y 224.636,Z 267.175,A -85,B 0,C 180,E1 -20942.265,E2 -20942.265} C_VEL
LIN {X 0,Y 224.605,Z 270.988,A -85,B 0,C 180,E1 -20943.006,E2 -20943.006} C_VEL
LIN {X 0,Y 223.724,Z 274.15,A -85,B 0,C 180,E1 -20943.557,E2 -20943.557} C_VEL
LIN {X 0,Y 220.964,Z 278.158,A -85,B 0,C 180,E1 -20944.143,E2 -20944.143} C_VEL
LIN {X 0,Y 216.15,Z 283.887,A -85,B 0,C 180,E1 -20945.047,E2 -20945.047} C_VEL
LIN {X 0,Y 214.651,Z 286.75,A -85,B 0,C 180,E1 -20945.693,E2 -20945.693} C_VEL
LIN {X 0,Y 212.111,Z 295.627,A -85,B 0,C 180,E1 -20948.293,E2 -20948.293} C_VEL
LIN {X 0,Y 209.723,Z 302.819,A -85,B 0,C 180,E1 -20950.929,E2 -20950.929} C_VEL
LIN {X 0,Y 208.073,Z 308.092,A -85,B 0,C 180,E1 -20953.315,E2 -20953.315} C_VEL
LIN {X 0,Y 206.429,Z 313.2,A -85,B 0,C 180,E1 -20956.212,E2 -20956.212} C_VEL
LIN {X 0,Y 205.394,Z 317.175,A -85,B 0,C 180,E1 -20959.152,E2 -20959.152} C_VEL
LIN {X 0,Y 204.679,Z 320.112,A -85,B 0,C 180,E1 -20962.105,E2 -20962.105} C_VEL
LIN {X 0,Y 204.347,Z 322.43,A -85,B 0,C 180,E1 -20965.856,E2 -20965.856} C_VEL
LIN {X 0,Y 204.363,Z 323.125,A -85,B 0,C 180,E1 -20968.029,E2 -20968.029} C_VEL
LIN {X 0,Y 204.451,Z 323.341,A -85,B 0,C 180,E1 -20970,E2 -20970} C_VEL
LIN {X 0,Y 204.364,Z 323.116,A -85,B 0,C 180,E1 -20971.97,E2 -20971.97} C_VEL
LIN {X 0,Y 204.358,Z 322.399,A -85,B 0,C 180,E1 -20974.186,E2 -20974.186} C_VEL
LIN {X 0,Y 204.679,Z 320.083,A -85,B 0,C 180,E1 -20977.894,E2 -20977.894} C_VEL
LIN {X 0,Y 205.393,Z 317.132,A -85,B 0,C 180,E1 -20980.847,E2 -20980.847} C_VEL
LIN {X 0,Y 206.428,Z 313.14,A -85,B 0,C 180,E1 -20983.787,E2 -20983.787} C_VEL
LIN {X 0,Y 208.366,Z 307.013,A -85,B 0,C 180,E1 -20987.165,E2 -20987.165} C_VEL
LIN {X 0,Y 210.542,Z 300.325,A -85,B 0,C 180,E1 -20990.007,E2 -20990.007} C_VEL
LIN {X 0,Y 212.674,Z 293.32,A -85,B 0,C 180,E1 -20992.403,E2 -20992.403} C_VEL
LIN {X 0,Y 214.99,Z 285.325,A -85,B 0,C 180,E1 -20994.632,E2 -20994.632} C_VEL
LIN {X 0,Y 217.819,Z 275.339,A -85,B 0,C 180,E1 -20996.853,E2 -20996.853} C_VEL
LIN {X 0,Y 218.071,Z 265.402,A -85,B 0,C 180,E1 -20998.908,E2 -20998.908} C_VEL
LIN {X 0,Y 217.461,Z 254.584,A -85,B 0,C 180,E1 -21000.867,E2 -21000.867} C_VEL
LIN {X 0,Y 215.964,Z 243.563,A -85,B 0,C 180,E1 -21002.644,E2 -21002.644} C_VEL
LIN {X 0,Y 213.469,Z 231.911,A -85,B 0,C 180,E1 -21004.343,E2 -21004.343} C_VEL
LIN {X 0,Y 210.132,Z 220.594,A -85,B 0,C 180,E1 -21005.865,E2 -21005.865} C_VEL
LIN {X 0,Y 208.841,Z 217.64,A -85,B 0,C 180,E1 -21006.308,E2 -21006.308} C_VEL
LIN {X 0,Y 208.602,Z 216.394,A -85,B 0,C 180,E1 -21006.449,E2 -21006.449} C_VEL
LIN {X 0,Y 208.671,Z 213.533,A -85,B 0,C 180,E1 -21009.785,E2 -21009.785} C_VEL
LIN {X 0,Y 208.362,Z 211.428,A -85,B 0,C 180,E1 -21012.422,E2 -21012.422} C_VEL
LIN {X 0,Y 207.689,Z 207.666,A -85,B 0,C 180,E1 -21017.407,E2 -21017.407} C_VEL
LIN {X 0,Y 207.12,Z 204.245,A -85,B 0,C 180,E1 -21022.354,E2 -21022.354} C_VEL
LIN {X 0,Y 206.7,Z 201.739,A -85,B 0,C 180,E1 -21026.46,E2 -21026.46} C_VEL
LIN {X 0,Y 206.735,Z 201.734,A -85,B 0,C 180,E1 -21031.58,E2 -21031.58} C_VEL
LIN {X 0,Y 206.753,Z 201.734,A -85,B 0,C 180,E1 -21036.604,E2 -21036.604} C_VEL
LIN {X 0,Y 206.872,Z 201.718,A -85,B 0,C 180,E1 -21042.196,E2 -21042.196} C_VEL
LIN {X 0,Y 206.894,Z 201.713,A -85,B 0,C 180,E1 -21046.244,E2 -21046.244} C_VEL
LIN {X 0,Y 207.077,Z 201.687,A -85,B 0,C 180,E1 -21050.23,E2 -21050.23} C_VEL
LIN {X 0,Y 207.045,Z 201.694,A -85,B 0,C 180,E1 -21054.155,E2 -21054.155} C_VEL
LIN {X 0,Y 207.377,Z 201.651,A -85,B 0,C 180,E1 -21058.058,E2 -21058.058} C_VEL
LIN {X 0,Y 207.514,Z 201.636,A -85,B 0,C 180,E1 -21060,E2 -21060} C_VEL
LIN {X 0,Y 207.377,Z 201.652,A -85,B 0,C 180,E1 -21061.942,E2 -21061.942} C_VEL
LIN {X 0,Y 207.128,Z 201.683,A -85,B 0,C 180,E1 -21067.801,E2 -21067.801} C_VEL
LIN {X 0,Y 206.923,Z 201.71,A -85,B 0,C 180,E1 -21071.759,E2 -21071.759} C_VEL
LIN {X 0,Y 206.866,Z 201.715,A -85,B 0,C 180,E1 -21075.771,E2 -21075.771} C_VEL
LIN {X 0,Y 206.783,Z 201.729,A -85,B 0,C 180,E1 -21079.869,E2 -21079.869} C_VEL
LIN {X 0,Y 206.763,Z 201.731,A -85,B 0,C 180,E1 -21084.072,E2 -21084.072} C_VEL
LIN {X 0,Y 206.743,Z 201.732,A -85,B 0,C 180,E1 -21088.419,E2 -21088.419} C_VEL
LIN {X 0,Y 206.697,Z 201.739,A -85,B 0,C 180,E1 -21092.958,E2 -21092.958} C_VEL
LIN {X 0,Y 206.673,Z 201.741,A -85,B 0,C 180,E1 -21097.742,E2 -21097.742} C_VEL
LIN {X 0,Y 206.64,Z 201.747,A -85,B 0,C 180,E1 -21101.563,E2 -21101.563} C_VEL
LIN {X 0,Y 206.625,Z 201.747,A -85,B 0,C 180,E1 -21104.417,E2 -21104.417} C_VEL
LIN {X 0,Y 206.98,Z 203.853,A -85,B 0,C 180,E1 -21108.332,E2 -21108.332} C_VEL
LIN {X 0,Y 207.159,Z 206.313,A -85,B 0,C 180,E1 -21112.363,E2 -21112.363} C_VEL
LIN {X 0,Y 207.162,Z 206.926,A -85,B 0,C 180,E1 -21113.326,E2 -21113.326} C_VEL
LIN {X 0,Y 208.376,Z 210.257,A -85,B 0,C 180,E1 -21113.823,E2 -21113.823} C_VEL
LIN {X 0,Y 212.229,Z 219.245,A -85,B 0,C 180,E1 -21115.274,E2 -21115.274} C_VEL
LIN {X 0,Y 215.286,Z 228.437,A -85,B 0,C 180,E1 -21116.774,E2 -21116.774} C_VEL
LIN {X 0,Y 218.041,Z 239.846,A -85,B 0,C 180,E1 -21118.733,E2 -21118.733} C_VEL
LIN {X 0,Y 219.738,Z 250.872,A -85,B 0,C 180,E1 -21120.821,E2 -21120.821} C_VEL
LIN {X 0,Y 220.17,Z 258.755,A -85,B 0,C 180,E1 -21122.429,E2 -21122.429} C_VEL
LIN {X 0,Y 217.836,Z 267.686,A -85,B 0,C 180,E1 -21124.18,E2 -21124.18} C_VEL
LIN {X 0,Y 215.3,Z 277.399,A -85,B 0,C 180,E1 -21126.607,E2 -21126.607} C_VEL
LIN {X 0,Y 212.613,Z 285.74,A -85,B 0,C 180,E1 -21129.186,E2 -21129.186} C_VEL
LIN {X 0,Y 210.158,Z 292.904,A -85,B 0,C 180,E1 -21131.981,E2 -21131.981} C_VEL
LIN {X 0,Y 208.523,Z 297.731,A -85,B 0,C 180,E1 -21134.358,E2 -21134.358} C_VEL
LIN {X 0,Y 206.923,Z 302.421,A -85,B 0,C 180,E1 -21137.246,E2 -21137.246} C_VEL
LIN {X 0,Y 205.822,Z 306.004,A -85,B 0,C 180,E1 -21140.17,E2 -21140.17} C_VEL
LIN {X 0,Y 205.276,Z 307.855,A -85,B 0,C 180,E1 -21142.129,E2 -21142.129} C_VEL
LIN {X 0,Y 204.901,Z 309.244,A -85,B 0,C 180,E1 -21144.094,E2 -21144.094} C_VEL
LIN {X 0,Y 204.524,Z 310.839,A -85,B 0,C 180,E1 -21148.031,E2 -21148.031} C_VEL
LIN {X 0,Y 204.503,Z 311.066,A -85,B 0,C 180,E1 -21150,E2 -21150} C_VEL
LIN {X 0,Y 204.523,Z 310.872,A -85,B 0,C 180,E1 -21151.97,E2 -21151.97} C_VEL
LIN {X 0,Y 204.901,Z 309.319,A -85,B 0,C 180,E1 -21155.907,E2 -21155.907} C_VEL
LIN {X 0,Y 205.276,Z 307.962,A -85,B 0,C 180,E1 -21157.872,E2 -21157.872} C_VEL
LIN {X 0,Y 206.106,Z 305.096,A -85,B 0,C 180,E1 -21160.81,E2 -21160.81} C_VEL
LIN {X 0,Y 207.356,Z 301.206,A -85,B 0,C 180,E1 -21163.725,E2 -21163.725} C_VEL
LIN {X 0,Y 209.091,Z 296.184,A -85,B 0,C 180,E1 -21166.601,E2 -21166.601} C_VEL
LIN {X 0,Y 211.246,Z 289.858,A -85,B 0,C 180,E1 -21169.433,E2 -21169.433} C_VEL
LIN {X 0,Y 213.947,Z 281.938,A -85,B 0,C 180,E1 -21172.196,E2 -21172.196} C_VEL
LIN {X 0,Y 216.328,Z 273.623,A -85,B 0,C 180,E1 -21174.542,E2 -21174.542} C_VEL
LIN {X 0,Y 218.898,Z 264.021,A -85,B 0,C 180,E1 -21176.711,E2 -21176.711} C_VEL
LIN {X 0,Y 220.277,Z 258.189,A -85,B 0,C 180,E1 -21177.815,E2 -21177.815} C_VEL
LIN {X 0,Y 219.425,Z 248.133,A -85,B 0,C 180,E1 -21179.861,E2 -21179.861} C_VEL
LIN {X 0,Y 217.717,Z 238.089,A -85,B 0,C 180,E1 -21181.717,E2 -21181.717} C_VEL
LIN {X 0,Y 215.014,Z 227.377,A -85,B 0,C 180,E1 -21183.541,E2 -21183.541} C_VEL
LIN {X 0,Y 211.23,Z 216.669,A -85,B 0,C 180,E1 -21185.291,E2 -21185.291} C_VEL
LIN {X 0,Y 208.082,Z 209.693,A -85,B 0,C 180,E1 -21186.433,E2 -21186.433} C_VEL
LIN {X 0,Y 207.148,Z 206.933,A -85,B 0,C 180,E1 -21186.835,E2 -21186.835} C_VEL
LIN {X 0,Y 207.049,Z 204.857,A -85,B 0,C 180,E1 -21190.161,E2 -21190.161} C_VEL
LIN {X 0,Y 206.73,Z 202.4,A -85,B 0,C 180,E1 -21194.445,E2 -21194.445} C_VEL
LIN {X 0,Y 206.628,Z 201.784,A -85,B 0,C 180,E1 -21195.584,E2 -21195.584} C_VEL
LIN {X 0,Y 206.661,Z 201.743,A -85,B 0,C 180,E1 -21199.748,E2 -21199.748} C_VEL
LIN {X 0,Y 206.701,Z 201.737,A -85,B 0,C 180,E1 -21204.689,E2 -21204.689} C_VEL
LIN {X 0,Y 206.709,Z 201.736,A -85,B 0,C 180,E1 -21209.336,E2 -21209.336} C_VEL
LIN {X 0,Y 206.734,Z 201.73,A -85,B 0,C 180,E1 -21213.772,E2 -21213.772} C_VEL
LIN {X 0,Y 206.76,Z 201.725,A -85,B 0,C 180,E1 -21218.043,E2 -21218.043} C_VEL
LIN {X 0,Y 206.876,Z 201.71,A -85,B 0,C 180,E1 -21222.197,E2 -21222.197} C_VEL
LIN {X 0,Y 206.897,Z 201.714,A -85,B 0,C 180,E1 -21226.244,E2 -21226.244} C_VEL
LIN {X 0,Y 207.081,Z 201.688,A -85,B 0,C 180,E1 -21230.23,E2 -21230.23} C_VEL
LIN {X 0,Y 207.049,Z 201.694,A -85,B 0,C 180,E1 -21234.155,E2 -21234.155} C_VEL
LIN {X 0,Y 207.379,Z 201.652,A -85,B 0,C 180,E1 -21238.058,E2 -21238.058} C_VEL
LIN {X 0,Y 207.517,Z 201.634,A -85,B 0,C 180,E1 -21240,E2 -21240} C_VEL
LIN {X 0,Y 207.38,Z 201.653,A -85,B 0,C 180,E1 -21241.942,E2 -21241.942} C_VEL
LIN {X 0,Y 207.127,Z 201.685,A -85,B 0,C 180,E1 -21247.8,E2 -21247.8} C_VEL
LIN {X 0,Y 206.933,Z 201.71,A -85,B 0,C 180,E1 -21251.758,E2 -21251.758} C_VEL
LIN {X 0,Y 206.869,Z 201.719,A -85,B 0,C 180,E1 -21255.77,E2 -21255.77} C_VEL
LIN {X 0,Y 206.78,Z 201.73,A -85,B 0,C 180,E1 -21259.869,E2 -21259.869} C_VEL
LIN {X 0,Y 206.749,Z 201.732,A -85,B 0,C 180,E1 -21264.074,E2 -21264.074} C_VEL
LIN {X 0,Y 206.738,Z 201.736,A -85,B 0,C 180,E1 -21268.42,E2 -21268.42} C_VEL
LIN {X 0,Y 206.693,Z 201.743,A -85,B 0,C 180,E1 -21273.541,E2 -21273.541} C_VEL
LIN {X 0,Y 207.166,Z 204.297,A -85,B 0,C 180,E1 -21277.636,E2 -21277.636} C_VEL
LIN {X 0,Y 207.692,Z 207.713,A -85,B 0,C 180,E1 -21282.592,E2 -21282.592} C_VEL
LIN {X 0,Y 208.361,Z 211.477,A -85,B 0,C 180,E1 -21287.577,E2 -21287.577} C_VEL
LIN {X 0,Y 208.682,Z 214.046,A -85,B 0,C 180,E1 -21290.769,E2 -21290.769} C_VEL
LIN {X 0,Y 208.64,Z 216.486,A -85,B 0,C 180,E1 -21293.533,E2 -21293.533} C_VEL
LIN {X 0,Y 209.592,Z 219.697,A -85,B 0,C 180,E1 -21293.913,E2 -21293.913} C_VEL
LIN {X 0,Y 212.18,Z 227.031,A -85,B 0,C 180,E1 -21294.937,E2 -21294.937} C_VEL
LIN {X 0,Y 215.232,Z 239.239,A -85,B 0,C 180,E1 -21296.663,E2 -21296.663} C_VEL
LIN {X 0,Y 217.139,Z 251.611,A -85,B 0,C 180,E1 -21298.584,E2 -21298.584} C_VEL
LIN {X 0,Y 217.985,Z 262.592,A -85,B 0,C 180,E1 -21300.517,E2 -21300.517} C_VEL
LIN {X 0,Y 217.973,Z 273.202,A -85,B 0,C 180,E1 -21302.648,E2 -21302.648} C_VEL
LIN {X 0,Y 217.626,Z 276.597,A -85,B 0,C 180,E1 -21303.379,E2 -21303.379} C_VEL
LIN {X 0,Y 214.651,Z 286.75,A -85,B 0,C 180,E1 -21305.693,E2 -21305.693} C_VEL
LIN {X 0,Y 212.848,Z 290.843,A -85,B 0,C 180,E1 -21306.731,E2 -21306.731} C_VEL
LIN {X 0,Y 208.274,Z 297.06,A -85,B 0,C 180,E1 -21308.429,E2 -21308.429} C_VEL
LIN {X 0,Y 203.728,Z 302.634,A -85,B 0,C 180,E1 -21310.334,E2 -21310.334} C_VEL
LIN {X 0,Y 202.01,Z 305.722,A -85,B 0,C 180,E1 -21311.676,E2 -21311.676} C_VEL
LIN {X 0,Y 200.022,Z 311.395,A -85,B 0,C 180,E1 -21314.72,E2 -21314.72} C_VEL
LIN {X 0,Y 198.705,Z 315.735,A -85,B 0,C 180,E1 -21317.747,E2 -21317.747} C_VEL
LIN {X 0,Y 198.091,Z 318.036,A -85,B 0,C 180,E1 -21319.782,E2 -21319.782} C_VEL
LIN {X 0,Y 197.646,Z 319.899,A -85,B 0,C 180,E1 -21321.822,E2 -21321.822} C_VEL
LIN {X 0,Y 197.368,Z 321.299,A -85,B 0,C 180,E1 -21323.867,E2 -21323.867} C_VEL
LIN {X 0,Y 197.244,Z 322.369,A -85,B 0,C 180,E1 -21326.087,E2 -21326.087} C_VEL
LIN {X 0,Y 197.352,Z 323.128,A -85,B 0,C 180,E1 -21330,E2 -21330} C_VEL
LIN {X 0,Y 197.245,Z 322.351,A -85,B 0,C 180,E1 -21333.918,E2 -21333.918} C_VEL
LIN {X 0,Y 197.368,Z 321.278,A -85,B 0,C 180,E1 -21336.132,E2 -21336.132} C_VEL
LIN {X 0,Y 197.645,Z 319.87,A -85,B 0,C 180,E1 -21338.177,E2 -21338.177} C_VEL
LIN {X 0,Y 198.381,Z 316.917,A -85,B 0,C 180,E1 -21341.235,E2 -21341.235} C_VEL
LIN {X 0,Y 199.495,Z 312.924,A -85,B 0,C 180,E1 -21344.276,E2 -21344.276} C_VEL
LIN {X 0,Y 201.58,Z 306.798,A -85,B 0,C 180,E1 -21347.762,E2 -21347.762} C_VEL
LIN {X 0,Y 203.882,Z 300.11,A -85,B 0,C 180,E1 -21350.69,E2 -21350.69} C_VEL
LIN {X 0,Y 206.448,Z 291.888,A -85,B 0,C 180,E1 -21353.55,E2 -21353.55} C_VEL
LIN {X 0,Y 209.115,Z 283.305,A -85,B 0,C 180,E1 -21355.906,E2 -21355.906} C_VEL
LIN {X 0,Y 211.185,Z 276.195,A -85,B 0,C 180,E1 -21357.499,E2 -21357.499} C_VEL
LIN {X 0,Y 211.521,Z 265.172,A -85,B 0,C 180,E1 -21359.893,E2 -21359.893} C_VEL
LIN {X 0,Y 210.92,Z 254.348,A -85,B 0,C 180,E1 -21361.935,E2 -21361.935} C_VEL
LIN {X 0,Y 209.395,Z 243.102,A -85,B 0,C 180,E1 -21363.831,E2 -21363.831} C_VEL
LIN {X 0,Y 207.008,Z 232.304,A -85,B 0,C 180,E1 -21365.511,E2 -21365.511} C_VEL
LIN {X 0,Y 204.503,Z 223.809,A -85,B 0,C 180,E1 -21366.771,E2 -21366.771} C_VEL
LIN {X 0,Y 202.575,Z 219.186,A -85,B 0,C 180,E1 -21367.501,E2 -21367.501} C_VEL
LIN {X 0,Y 201.671,Z 216.139,A -85,B 0,C 180,E1 -21367.917,E2 -21367.917} C_VEL
LIN {X 0,Y 201.457,Z 213.277,A -85,B 0,C 180,E1 -21371.515,E2 -21371.515} C_VEL
LIN {X 0,Y 200.935,Z 210.235,A -85,B 0,C 180,E1 -21375.611,E2 -21375.611} C_VEL
LIN {X 0,Y 200.339,Z 206.855,A -85,B 0,C 180,E1 -21380.512,E2 -21380.512} C_VEL
LIN {X 0,Y 199.861,Z 203.58,A -85,B 0,C 180,E1 -21385.762,E2 -21385.762} C_VEL
LIN {X 0,Y 199.651,Z 202.617,A -85,B 0,C 180,E1 -21387.653,E2 -21387.653} C_VEL
LIN {X 0,Y 199.684,Z 202.613,A -85,B 0,C 180,E1 -21392.771,E2 -21392.771} C_VEL
LIN {X 0,Y 199.713,Z 202.611,A -85,B 0,C 180,E1 -21397.226,E2 -21397.226} C_VEL
LIN {X 0,Y 199.795,Z 202.599,A -85,B 0,C 180,E1 -21401.758,E2 -21401.758} C_VEL
LIN {X 0,Y 199.834,Z 202.592,A -85,B 0,C 180,E1 -21405.748,E2 -21405.748} C_VEL
LIN {X 0,Y 200.021,Z 202.564,A -85,B 0,C 180,E1 -21409.882,E2 -21409.882} C_VEL
LIN {X 0,Y 200.007,Z 202.571,A -85,B 0,C 180,E1 -21413.949,E2 -21413.949} C_VEL
LIN {X 0,Y 200.316,Z 202.531,A -85,B 0,C 180,E1 -21417.989,E2 -21417.989} C_VEL
LIN {X 0,Y 200.478,Z 202.512,A -85,B 0,C 180,E1 -21420,E2 -21420} C_VEL
LIN {X 0,Y 200.015,Z 202.568,A -85,B 0,C 180,E1 -21424.03,E2 -21424.03} C_VEL
LIN {X 0,Y 200.075,Z 202.562,A -85,B 0,C 180,E1 -21428.077,E2 -21428.077} C_VEL
LIN {X 0,Y 199.873,Z 202.588,A -85,B 0,C 180,E1 -21432.18,E2 -21432.18} C_VEL
LIN {X 0,Y 199.803,Z 202.597,A -85,B 0,C 180,E1 -21436.344,E2 -21436.344} C_VEL
LIN {X 0,Y 199.699,Z 202.607,A -85,B 0,C 180,E1 -21440.606,E2 -21440.606} C_VEL
LIN {X 0,Y 199.672,Z 202.613,A -85,B 0,C 180,E1 -21444.985,E2 -21444.985} C_VEL
LIN {X 0,Y 199.67,Z 202.613,A -85,B 0,C 180,E1 -21449.523,E2 -21449.523} C_VEL
LIN {X 0,Y 199.67,Z 202.614,A -85,B 0,C 180,E1 -21452.356,E2 -21452.356} C_VEL
LIN {X 0,Y 199.619,Z 202.619,A -85,B 0,C 180,E1 -21456.764,E2 -21456.764} C_VEL
LIN {X 0,Y 199.605,Z 202.623,A -85,B 0,C 180,E1 -21459.329,E2 -21459.329} C_VEL
LIN {X 0,Y 199.572,Z 202.626,A -85,B 0,C 180,E1 -21462.31,E2 -21462.31} C_VEL
LIN {X 0,Y 199.718,Z 203.475,A -85,B 0,C 180,E1 -21465.269,E2 -21465.269} C_VEL
LIN {X 0,Y 199.993,Z 205.002,A -85,B 0,C 180,E1 -21468.112,E2 -21468.112} C_VEL
LIN {X 0,Y 200.204,Z 207.379,A -85,B 0,C 180,E1 -21471.876,E2 -21471.876} C_VEL
LIN {X 0,Y 201.364,Z 210.456,A -85,B 0,C 180,E1 -21472.344,E2 -21472.344} C_VEL
LIN {X 0,Y 202.674,Z 213.062,A -85,B 0,C 180,E1 -21472.813,E2 -21472.813} C_VEL
LIN {X 0,Y 206.565,Z 222.361,A -85,B 0,C 180,E1 -21474.465,E2 -21474.465} C_VEL
LIN {X 0,Y 209.511,Z 231.751,A -85,B 0,C 180,E1 -21476.122,E2 -21476.122} C_VEL
LIN {X 0,Y 211.953,Z 242.767,A -85,B 0,C 180,E1 -21478.161,E2 -21478.161} C_VEL
LIN {X 0,Y 213.432,Z 253.846,A -85,B 0,C 180,E1 -21480.402,E2 -21480.402} C_VEL
LIN {X 0,Y 213.616,Z 260.153,A -85,B 0,C 180,E1 -21481.775,E2 -21481.775} C_VEL
LIN {X 0,Y 210.917,Z 269.855,A -85,B 0,C 180,E1 -21483.801,E2 -21483.801} C_VEL
LIN {X 0,Y 208.434,Z 278.674,A -85,B 0,C 180,E1 -21486.133,E2 -21486.133} C_VEL
LIN {X 0,Y 205.549,Z 287.281,A -85,B 0,C 180,E1 -21488.961,E2 -21488.961} C_VEL
LIN {X 0,Y 203.024,Z 294.145,A -85,B 0,C 180,E1 -21491.848,E2 -21491.848} C_VEL
LIN {X 0,Y 201.086,Z 299.635,A -85,B 0,C 180,E1 -21494.804,E2 -21494.804} C_VEL
LIN {X 0,Y 199.534,Z 303.943,A -85,B 0,C 180,E1 -21497.8,E2 -21497.8} C_VEL
LIN {X 0,Y 198.817,Z 306.219,A -85,B 0,C 180,E1 -21499.82,E2 -21499.82} C_VEL
LIN {X 0,Y 198.24,Z 308.069,A -85,B 0,C 180,E1 -21501.848,E2 -21501.848} C_VEL
LIN {X 0,Y 197.765,Z 309.682,A -85,B 0,C 180,E1 -21504.294,E2 -21504.294} C_VEL
LIN {X 0,Y 197.43,Z 311.052,A -85,B 0,C 180,E1 -21507.96,E2 -21507.96} C_VEL
LIN {X 0,Y 197.424,Z 311.278,A -85,B 0,C 180,E1 -21510,E2 -21510} C_VEL
LIN {X 0,Y 197.429,Z 311.085,A -85,B 0,C 180,E1 -21512.041,E2 -21512.041} C_VEL
LIN {X 0,Y 197.834,Z 309.532,A -85,B 0,C 180,E1 -21516.118,E2 -21516.118} C_VEL
LIN {X 0,Y 198.24,Z 308.175,A -85,B 0,C 180,E1 -21518.153,E2 -21518.153} C_VEL
LIN {X 0,Y 199.138,Z 305.308,A -85,B 0,C 180,E1 -21521.193,E2 -21521.193} C_VEL
LIN {X 0,Y 200.468,Z 301.418,A -85,B 0,C 180,E1 -21524.206,E2 -21524.206} C_VEL
LIN {X 0,Y 202.283,Z 296.396,A -85,B 0,C 180,E1 -21527.177,E2 -21527.177} C_VEL
LIN {X 0,Y 204.579,Z 290.068,A -85,B 0,C 180,E1 -21530.093,E2 -21530.093} C_VEL
LIN {X 0,Y 207.393,Z 282.148,A -85,B 0,C 180,E1 -21532.937,E2 -21532.937} C_VEL
LIN {X 0,Y 210.02,Z 273.376,A -85,B 0,C 180,E1 -21535.467,E2 -21535.467} C_VEL
LIN {X 0,Y 212.598,Z 264.23,A -85,B 0,C 180,E1 -21537.569,E2 -21537.569} C_VEL
LIN {X 0,Y 213.761,Z 259.62,A -85,B 0,C 180,E1 -21538.472,E2 -21538.472} C_VEL
LIN {X 0,Y 213.108,Z 250.453,A -85,B 0,C 180,E1 -21540.455,E2 -21540.455} C_VEL
LIN {X 0,Y 211.58,Z 240.498,A -85,B 0,C 180,E1 -21542.42,E2 -21542.42} C_VEL
LIN {X 0,Y 208.85,Z 229.351,A -85,B 0,C 180,E1 -21544.469,E2 -21544.469} C_VEL
LIN {X 0,Y 204.979,Z 218.129,A -85,B 0,C 180,E1 -21546.433,E2 -21546.433} C_VEL
LIN {X 0,Y 201.598,Z 210.793,A -85,B 0,C 180,E1 -21547.744,E2 -21547.744} C_VEL
LIN {X 0,Y 200.259,Z 207.702,A -85,B 0,C 180,E1 -21548.258,E2 -21548.258} C_VEL
LIN {X 0,Y 200.167,Z 207.188,A -85,B 0,C 180,E1 -21548.327,E2 -21548.327} C_VEL
LIN {X 0,Y 199.914,Z 204.82,A -85,B 0,C 180,E1 -21552.416,E2 -21552.416} C_VEL
LIN {X 0,Y 199.69,Z 203.296,A -85,B 0,C 180,E1 -21555.26,E2 -21555.26} C_VEL
LIN {X 0,Y 199.58,Z 202.625,A -85,B 0,C 180,E1 -21558.005,E2 -21558.005} C_VEL
LIN {X 0,Y 199.609,Z 202.62,A -85,B 0,C 180,E1 -21560.769,E2 -21560.769} C_VEL
LIN {X 0,Y 199.613,Z 202.62,A -85,B 0,C 180,E1 -21565.713,E2 -21565.713} C_VEL
LIN {X 0,Y 199.695,Z 202.608,A -85,B 0,C 180,E1 -21568.136,E2 -21568.136} C_VEL
LIN {X 0,Y 199.688,Z 202.61,A -85,B 0,C 180,E1 -21572.772,E2 -21572.772} C_VEL
LIN {X 0,Y 199.74,Z 202.601,A -85,B 0,C 180,E1 -21577.229,E2 -21577.229} C_VEL
LIN {X 0,Y 199.799,Z 202.592,A -85,B 0,C 180,E1 -21581.758,E2 -21581.758} C_VEL
LIN {X 0,Y 199.838,Z 202.592,A -85,B 0,C 180,E1 -21585.748,E2 -21585.748} C_VEL
LIN {X 0,Y 200.024,Z 202.568,A -85,B 0,C 180,E1 -21589.882,E2 -21589.882} C_VEL
LIN {X 0,Y 200.012,Z 202.571,A -85,B 0,C 180,E1 -21593.949,E2 -21593.949} C_VEL
LIN {X 0,Y 200.318,Z 202.531,A -85,B 0,C 180,E1 -21597.989,E2 -21597.989} C_VEL
LIN {X 0,Y 200.481,Z 202.51,A -85,B 0,C 180,E1 -21600,E2 -21600} C_VEL
LIN {X 0,Y 200.018,Z 202.571,A -85,B 0,C 180,E1 -21604.03,E2 -21604.03} C_VEL
LIN {X 0,Y 200.075,Z 202.564,A -85,B 0,C 180,E1 -21608.077,E2 -21608.077} C_VEL
LIN {X 0,Y 199.881,Z 202.588,A -85,B 0,C 180,E1 -21612.179,E2 -21612.179} C_VEL
LIN {X 0,Y 199.807,Z 202.598,A -85,B 0,C 180,E1 -21616.343,E2 -21616.343} C_VEL
LIN {X 0,Y 199.693,Z 202.611,A -85,B 0,C 180,E1 -21620.606,E2 -21620.606} C_VEL
LIN {X 0,Y 199.666,Z 202.615,A -85,B 0,C 180,E1 -21624.985,E2 -21624.985} C_VEL
LIN {X 0,Y 199.666,Z 202.617,A -85,B 0,C 180,E1 -21629.524,E2 -21629.524} C_VEL
LIN {X 0,Y 199.681,Z 202.754,A -85,B 0,C 180,E1 -21632.687,E2 -21632.687} C_VEL
LIN {X 0,Y 200.069,Z 205.094,A -85,B 0,C 180,E1 -21636.668,E2 -21636.668} C_VEL
LIN {X 0,Y 200.62,Z 208.421,A -85,B 0,C 180,E1 -21641.728,E2 -21641.728} C_VEL
LIN {X 0,Y 201.078,Z 211.211,A -85,B 0,C 180,E1 -21645.65,E2 -21645.65} C_VEL
LIN {X 0,Y 201.634,Z 214.554,A -85,B 0,C 180,E1 -21650.069,E2 -21650.069} C_VEL
LIN {X 0,Y 201.639,Z 216.158,A -85,B 0,C 180,E1 -21652.041,E2 -21652.041} C_VEL
LIN {X 0,Y 202.763,Z 219.539,A -85,B 0,C 180,E1 -21652.499,E2 -21652.499} C_VEL
LIN {X 0,Y 205.821,Z 227.605,A -85,B 0,C 180,E1 -21653.751,E2 -21653.751} C_VEL
LIN {X 0,Y 208.799,Z 239.527,A -85,B 0,C 180,E1 -21655.552,E2 -21655.552} C_VEL
LIN {X 0,Y 210.628,Z 251.387,A -85,B 0,C 180,E1 -21657.495,E2 -21657.495} C_VEL
LIN {X 0,Y 211.478,Z 261.967,A -85,B 0,C 180,E1 -21659.438,E2 -21659.438} C_VEL
LIN {X 0,Y 211.4,Z 272.991,A -85,B 0,C 180,E1 -21661.724,E2 -21661.724} C_VEL
LIN {X 0,Y 210.973,Z 277.459,A -85,B 0,C 180,E1 -21662.739,E2 -21662.739} C_VEL
LIN {X 0,Y 208.021,Z 287.088,A -85,B 0,C 180,E1 -21665.03,E2 -21665.03} C_VEL
LIN {X 0,Y 205.613,Z 294.829,A -85,B 0,C 180,E1 -21667.351,E2 -21667.351} C_VEL
LIN {X 0,Y 203.426,Z 301.451,A -85,B 0,C 180,E1 -21669.788,E2 -21669.788} C_VEL
LIN {X 0,Y 202.01,Z 305.722,A -85,B 0,C 180,E1 -21671.676,E2 -21671.676} C_VEL
LIN {X 0,Y 200.362,Z 308.604,A -85,B 0,C 180,E1 -21673.074,E2 -21673.074} C_VEL
LIN {X 0,Y 196.173,Z 312.79,A -85,B 0,C 180,E1 -21675.374,E2 -21675.374} C_VEL
LIN {X 0,Y 192.245,Z 316.24,A -85,B 0,C 180,E1 -21677.862,E2 -21677.862} C_VEL
LIN {X 0,Y 191.046,Z 317.925,A -85,B 0,C 180,E1 -21679.518,E2 -21679.518} C_VEL
LIN {X 0,Y 190.588,Z 319.686,A -85,B 0,C 180,E1 -21681.517,E2 -21681.517} C_VEL
LIN {X 0,Y 190.3,Z 321.086,A -85,B 0,C 180,E1 -21683.638,E2 -21683.638} C_VEL
LIN {X 0,Y 190.136,Z 322.323,A -85,B 0,C 180,E1 -21686.378,E2 -21686.378} C_VEL
LIN {X 0,Y 190.256,Z 322.915,A -85,B 0,C 180,E1 -21689.999,E2 -21689.999} C_VEL
LIN {X 0,Y 190.137,Z 322.305,A -85,B 0,C 180,E1 -21693.627,E2 -21693.627} C_VEL
LIN {X 0,Y 190.3,Z 321.064,A -85,B 0,C 180,E1 -21696.361,E2 -21696.361} C_VEL
LIN {X 0,Y 190.587,Z 319.655,A -85,B 0,C 180,E1 -21698.482,E2 -21698.482} C_VEL
LIN {X 0,Y 191.381,Z 316.702,A -85,B 0,C 180,E1 -21701.652,E2 -21701.652} C_VEL
LIN {X 0,Y 192.583,Z 312.709,A -85,B 0,C 180,E1 -21704.8,E2 -21704.8} C_VEL
LIN {X 0,Y 194.816,Z 306.582,A -85,B 0,C 180,E1 -21708.4,E2 -21708.4} C_VEL
LIN {X 0,Y 197.251,Z 299.894,A -85,B 0,C 180,E1 -21711.42,E2 -21711.42} C_VEL
LIN {X 0,Y 199.939,Z 291.594,A -85,B 0,C 180,E1 -21714.393,E2 -21714.393} C_VEL
LIN {X 0,Y 202.73,Z 283.088,A -85,B 0,C 180,E1 -21716.786,E2 -21716.786} C_VEL
LIN {X 0,Y 204.58,Z 277.05,A -85,B 0,C 180,E1 -21718.187,E2 -21718.187} C_VEL
LIN {X 0,Y 205.031,Z 266.171,A -85,B 0,C 180,E1 -21720.678,E2 -21720.678} C_VEL
LIN {X 0,Y 204.624,Z 256.348,A -85,B 0,C 180,E1 -21722.654,E2 -21722.654} C_VEL
LIN {X 0,Y 203.153,Z 244.226,A -85,B 0,C 180,E1 -21724.839,E2 -21724.839} C_VEL
LIN {X 0,Y 200.595,Z 232.45,A -85,B 0,C 180,E1 -21726.789,E2 -21726.789} C_VEL
LIN {X 0,Y 197.97,Z 224.133,A -85,B 0,C 180,E1 -21728.146,E2 -21728.146} C_VEL
LIN {X 0,Y 195.826,Z 219.346,A -85,B 0,C 180,E1 -21729.001,E2 -21729.001} C_VEL
LIN {X 0,Y 194.643,Z 215.903,A -85,B 0,C 180,E1 -21729.53,E2 -21729.53} C_VEL
LIN {X 0,Y 194.174,Z 212.88,A -85,B 0,C 180,E1 -21733.624,E2 -21733.624} C_VEL
LIN {X 0,Y 193.822,Z 210.882,A -85,B 0,C 180,E1 -21736.485,E2 -21736.485} C_VEL
LIN {X 0,Y 193.429,Z 208.72,A -85,B 0,C 180,E1 -21739.729,E2 -21739.729} C_VEL
LIN {X 0,Y 192.999,Z 205.868,A -85,B 0,C 180,E1 -21744.364,E2 -21744.364} C_VEL
LIN {X 0,Y 192.619,Z 203.493,A -85,B 0,C 180,E1 -21748.702,E2 -21748.702} C_VEL
LIN {X 0,Y 192.659,Z 203.488,A -85,B 0,C 180,E1 -21751.691,E2 -21751.691} C_VEL
LIN {X 0,Y 192.684,Z 203.486,A -85,B 0,C 180,E1 -21756.346,E2 -21756.346} C_VEL
LIN {X 0,Y 192.73,Z 203.479,A -85,B 0,C 180,E1 -21761.458,E2 -21761.458} C_VEL
LIN {X 0,Y 192.762,Z 203.475,A -85,B 0,C 180,E1 -21765.214,E2 -21765.214} C_VEL
LIN {X 0,Y 192.944,Z 203.444,A -85,B 0,C 180,E1 -21769.567,E2 -21769.567} C_VEL
LIN {X 0,Y 192.97,Z 203.448,A -85,B 0,C 180,E1 -21773.727,E2 -21773.727} C_VEL
LIN {X 0,Y 193.257,Z 203.41,A -85,B 0,C 180,E1 -21777.916,E2 -21777.916} C_VEL
LIN {X 0,Y 193.442,Z 203.389,A -85,B 0,C 180,E1 -21780,E2 -21780} C_VEL
LIN {X 0,Y 192.961,Z 203.447,A -85,B 0,C 180,E1 -21784.177,E2 -21784.177} C_VEL
LIN {X 0,Y 193.025,Z 203.442,A -85,B 0,C 180,E1 -21788.374,E2 -21788.374} C_VEL
LIN {X 0,Y 192.801,Z 203.467,A -85,B 0,C 180,E1 -21792.634,E2 -21792.634} C_VEL
LIN {X 0,Y 192.757,Z 203.474,A -85,B 0,C 180,E1 -21796.959,E2 -21796.959} C_VEL
LIN {X 0,Y 192.636,Z 203.488,A -85,B 0,C 180,E1 -21801.398,E2 -21801.398} C_VEL
LIN {X 0,Y 192.663,Z 203.487,A -85,B 0,C 180,E1 -21804.225,E2 -21804.225} C_VEL
LIN {X 0,Y 192.648,Z 203.488,A -85,B 0,C 180,E1 -21808.892,E2 -21808.892} C_VEL
LIN {X 0,Y 192.596,Z 203.495,A -85,B 0,C 180,E1 -21813.187,E2 -21813.187} C_VEL
LIN {X 0,Y 192.548,Z 203.504,A -85,B 0,C 180,E1 -21818.353,E2 -21818.353} C_VEL
LIN {X 0,Y 192.557,Z 203.755,A -85,B 0,C 180,E1 -21823.118,E2 -21823.118} C_VEL
LIN {X 0,Y 192.844,Z 205.617,A -85,B 0,C 180,E1 -21826.793,E2 -21826.793} C_VEL
LIN {X 0,Y 193.096,Z 207.438,A -85,B 0,C 180,E1 -21830.174,E2 -21830.174} C_VEL
LIN {X 0,Y 194.331,Z 210.647,A -85,B 0,C 180,E1 -21830.719,E2 -21830.719} C_VEL
LIN {X 0,Y 195.581,Z 212.828,A -85,B 0,C 180,E1 -21831.18,E2 -21831.18} C_VEL
LIN {X 0,Y 200.019,Z 222.998,A -85,B 0,C 180,E1 -21833.154,E2 -21833.154} C_VEL
LIN {X 0,Y 203.371,Z 233.594,A -85,B 0,C 180,E1 -21835.17,E2 -21835.17} C_VEL
LIN {X 0,Y 205.611,Z 244.168,A -85,B 0,C 180,E1 -21837.251,E2 -21837.251} C_VEL
LIN {X 0,Y 206.888,Z 254.078,A -85,B 0,C 180,E1 -21839.367,E2 -21839.367} C_VEL
LIN {X 0,Y 207.06,Z 261.54,A -85,B 0,C 180,E1 -21841.075,E2 -21841.075} C_VEL
LIN {X 0,Y 204.564,Z 270.072,A -85,B 0,C 180,E1 -21842.922,E2 -21842.922} C_VEL
LIN {X 0,Y 201.949,Z 278.89,A -85,B 0,C 180,E1 -21845.317,E2 -21845.317} C_VEL
LIN {X 0,Y 198.946,Z 287.496,A -85,B 0,C 180,E1 -21848.228,E2 -21848.228} C_VEL
LIN {X 0,Y 196.278,Z 294.36,A -85,B 0,C 180,E1 -21851.201,E2 -21851.201} C_VEL
LIN {X 0,Y 194.237,Z 299.85,A -85,B 0,C 180,E1 -21854.255,E2 -21854.255} C_VEL
LIN {X 0,Y 192.606,Z 304.157,A -85,B 0,C 180,E1 -21857.354,E2 -21857.354} C_VEL
LIN {X 0,Y 191.837,Z 306.433,A -85,B 0,C 180,E1 -21859.446,E2 -21859.446} C_VEL
LIN {X 0,Y 191.208,Z 308.283,A -85,B 0,C 180,E1 -21861.546,E2 -21861.546} C_VEL
LIN {X 0,Y 190.643,Z 310.102,A -85,B 0,C 180,E1 -21864.473,E2 -21864.473} C_VEL
LIN {X 0,Y 190.339,Z 311.265,A -85,B 0,C 180,E1 -21867.884,E2 -21867.884} C_VEL
LIN {X 0,Y 190.328,Z 311.492,A -85,B 0,C 180,E1 -21870.001,E2 -21870.001} C_VEL
LIN {X 0,Y 190.339,Z 311.297,A -85,B 0,C 180,E1 -21872.117,E2 -21872.117} C_VEL
LIN {X 0,Y 190.779,Z 309.744,A -85,B 0,C 180,E1 -21876.346,E2 -21876.346} C_VEL
LIN {X 0,Y 191.207,Z 308.387,A -85,B 0,C 180,E1 -21878.455,E2 -21878.455} C_VEL
LIN {X 0,Y 192.165,Z 305.52,A -85,B 0,C 180,E1 -21881.605,E2 -21881.605} C_VEL
LIN {X 0,Y 193.599,Z 301.629,A -85,B 0,C 180,E1 -21884.721,E2 -21884.721} C_VEL
LIN {X 0,Y 195.502,Z 296.608,A -85,B 0,C 180,E1 -21887.792,E2 -21887.792} C_VEL
LIN {X 0,Y 197.927,Z 290.279,A -85,B 0,C 180,E1 -21890.799,E2 -21890.799} C_VEL
LIN {X 0,Y 200.878,Z 282.358,A -85,B 0,C 180,E1 -21893.725,E2 -21893.725} C_VEL
LIN {X 0,Y 203.543,Z 273.857,A -85,B 0,C 180,E1 -21896.254,E2 -21896.254} C_VEL
LIN {X 0,Y 206.35,Z 264.439,A -85,B 0,C 180,E1 -21898.478,E2 -21898.478} C_VEL
LIN {X 0,Y 207.241,Z 260.999,A -85,B 0,C 180,E1 -21899.176,E2 -21899.176} C_VEL
LIN {X 0,Y 206.613,Z 251.28,A -85,B 0,C 180,E1 -21901.397,E2 -21901.397} C_VEL
LIN {X 0,Y 205.229,Z 241.813,A -85,B 0,C 180,E1 -21903.37,E2 -21903.37} C_VEL
LIN {X 0,Y 202.723,Z 231.218,A -85,B 0,C 180,E1 -21905.444,E2 -21905.444} C_VEL
LIN {X 0,Y 199.385,Z 221.408,A -85,B 0,C 180,E1 -21907.317,E2 -21907.317} C_VEL
LIN {X 0,Y 195.04,Z 211.67,A -85,B 0,C 180,E1 -21909.204,E2 -21909.204} C_VEL
LIN {X 0,Y 193.334,Z 208.549,A -85,B 0,C 180,E1 -21909.855,E2 -21909.855} C_VEL
LIN {X 0,Y 193.066,Z 207.42,A -85,B 0,C 180,E1 -21910.033,E2 -21910.033} C_VEL
LIN {X 0,Y 192.787,Z 205.369,A -85,B 0,C 180,E1 -21913.84,E2 -21913.84} C_VEL
LIN {X 0,Y 192.56,Z 203.849,A -85,B 0,C 180,E1 -21916.883,E2 -21916.883} C_VEL
LIN {X 0,Y 192.517,Z 203.505,A -85,B 0,C 180,E1 -21920.052,E2 -21920.052} C_VEL
LIN {X 0,Y 192.561,Z 203.5,A -85,B 0,C 180,E1 -21924.27,E2 -21924.27} C_VEL
LIN {X 0,Y 192.609,Z 203.491,A -85,B 0,C 180,E1 -21927.06,E2 -21927.06} C_VEL
LIN {X 0,Y 192.663,Z 203.485,A -85,B 0,C 180,E1 -21931.691,E2 -21931.691} C_VEL
LIN {X 0,Y 192.708,Z 203.48,A -85,B 0,C 180,E1 -21936.349,E2 -21936.349} C_VEL
LIN {X 0,Y 192.734,Z 203.472,A -85,B 0,C 180,E1 -21941.457,E2 -21941.457} C_VEL
LIN {X 0,Y 192.766,Z 203.473,A -85,B 0,C 180,E1 -21945.214,E2 -21945.214} C_VEL
LIN {X 0,Y 192.947,Z 203.451,A -85,B 0,C 180,E1 -21949.567,E2 -21949.567} C_VEL
LIN {X 0,Y 192.975,Z 203.448,A -85,B 0,C 180,E1 -21953.727,E2 -21953.727} C_VEL
LIN {X 0,Y 193.26,Z 203.411,A -85,B 0,C 180,E1 -21957.916,E2 -21957.916} C_VEL
LIN {X 0,Y 193.445,Z 203.387,A -85,B 0,C 180,E1 -21960,E2 -21960} C_VEL
LIN {X 0,Y 192.964,Z 203.45,A -85,B 0,C 180,E1 -21964.177,E2 -21964.177} C_VEL
LIN {X 0,Y 193.026,Z 203.443,A -85,B 0,C 180,E1 -21968.374,E2 -21968.374} C_VEL
LIN {X 0,Y 192.807,Z 203.471,A -85,B 0,C 180,E1 -21972.633,E2 -21972.633} C_VEL
LIN {X 0,Y 192.76,Z 203.476,A -85,B 0,C 180,E1 -21976.958,E2 -21976.958} C_VEL
LIN {X 0,Y 192.624,Z 203.492,A -85,B 0,C 180,E1 -21981.399,E2 -21981.399} C_VEL
LIN {X 0,Y 192.649,Z 203.488,A -85,B 0,C 180,E1 -21984.213,E2 -21984.213} C_VEL
LIN {X 0,Y 192.646,Z 203.49,A -85,B 0,C 180,E1 -21988.889,E2 -21988.889} C_VEL
LIN {X 0,Y 192.622,Z 203.519,A -85,B 0,C 180,E1 -21991.297,E2 -21991.297} C_VEL
LIN {X 0,Y 193.022,Z 205.917,A -85,B 0,C 180,E1 -21995.631,E2 -21995.631} C_VEL
LIN {X 0,Y 193.501,Z 209.142,A -85,B 0,C 180,E1 -22000.826,E2 -22000.826} C_VEL
LIN {X 0,Y 193.827,Z 210.956,A -85,B 0,C 180,E1 -22003.545,E2 -22003.545} C_VEL
LIN {X 0,Y 194.381,Z 214.123,A -85,B 0,C 180,E1 -22008.02,E2 -22008.02} C_VEL
LIN {X 0,Y 194.628,Z 215.949,A -85,B 0,C 180,E1 -22010.417,E2 -22010.417} C_VEL
LIN {X 0,Y 195.738,Z 219.238,A -85,B 0,C 180,E1 -22010.9,E2 -22010.9} C_VEL
LIN {X 0,Y 196.797,Z 221.363,A -85,B 0,C 180,E1 -22011.3,E2 -22011.3} C_VEL
LIN {X 0,Y 200.271,Z 230.917,A -85,B 0,C 180,E1 -22012.92,E2 -22012.92} C_VEL
LIN {X 0,Y 202.869,Z 242.26,A -85,B 0,C 180,E1 -22014.784,E2 -22014.784} C_VEL
LIN {X 0,Y 204.299,Z 252.658,A -85,B 0,C 180,E1 -22016.604,E2 -22016.604} C_VEL
LIN {X 0,Y 205.024,Z 262.947,A -85,B 0,C 180,E1 -22018.607,E2 -22018.607} C_VEL
LIN {X 0,Y 204.842,Z 274.077,A -85,B 0,C 180,E1 -22021.042,E2 -22021.042} C_VEL
LIN {X 0,Y 204.346,Z 278.321,A -85,B 0,C 180,E1 -22022.056,E2 -22022.056} C_VEL
LIN {X 0,Y 201.583,Z 286.841,A -85,B 0,C 180,E1 -22024.163,E2 -22024.163} C_VEL
LIN {X 0,Y 198.813,Z 295.289,A -85,B 0,C 180,E1 -22026.795,E2 -22026.795} C_VEL
LIN {X 0,Y 196.31,Z 302.395,A -85,B 0,C 180,E1 -22029.57,E2 -22029.57} C_VEL
LIN {X 0,Y 193.778,Z 309.489,A -85,B 0,C 180,E1 -22033.133,E2 -22033.133} C_VEL
LIN {X 0,Y 192.164,Z 314.211,A -85,B 0,C 180,E1 -22036.247,E2 -22036.247} C_VEL
LIN {X 0,Y 191.046,Z 317.925,A -85,B 0,C 180,E1 -22039.518,E2 -22039.518} C_VEL
LIN {X 0,Y 189.97,Z 319.444,A -85,B 0,C 180,E1 -22041.214,E2 -22041.214} C_VEL
LIN {X 0,Y 186.709,Z 321.239,A -85,B 0,C 180,E1 -22044.011,E2 -22044.011} C_VEL
LIN {X 0,Y 184.172,Z 322.169,A -85,B 0,C 180,E1 -22046.331,E2 -22046.331} C_VEL
LIN {X 0,Y 183.143,Z 322.563,A -85,B 0,C 180,E1 -22048.154,E2 -22048.154} C_VEL
LIN {X 0,Y 183.079,Z 322.582,A -85,B 0,C 180,E1 -22048.774,E2 -22048.774} C_VEL
LIN {X 0,Y 183.163,Z 322.702,A -85,B 0,C 180,E1 -22049.999,E2 -22049.999} C_VEL
LIN {X 0,Y 183.053,Z 322.205,A -85,B 0,C 180,E1 -22053.413,E2 -22053.413} C_VEL
LIN {X 0,Y 183.229,Z 320.85,A -85,B 0,C 180,E1 -22056.607,E2 -22056.607} C_VEL
LIN {X 0,Y 183.551,Z 319.44,A -85,B 0,C 180,E1 -22058.809,E2 -22058.809} C_VEL
LIN {X 0,Y 184.404,Z 316.487,A -85,B 0,C 180,E1 -22062.099,E2 -22062.099} C_VEL
LIN {X 0,Y 185.689,Z 312.494,A -85,B 0,C 180,E1 -22065.363,E2 -22065.363} C_VEL
LIN {X 0,Y 188.073,Z 306.367,A -85,B 0,C 180,E1 -22069.085,E2 -22069.085} C_VEL
LIN {X 0,Y 190.613,Z 299.77,A -85,B 0,C 180,E1 -22072.162,E2 -22072.162} C_VEL
LIN {X 0,Y 193.461,Z 291.378,A -85,B 0,C 180,E1 -22075.267,E2 -22075.267} C_VEL
LIN {X 0,Y 196.403,Z 282.871,A -85,B 0,C 180,E1 -22077.722,E2 -22077.722} C_VEL
LIN {X 0,Y 198.001,Z 277.905,A -85,B 0,C 180,E1 -22078.921,E2 -22078.921} C_VEL
LIN {X 0,Y 198.584,Z 267.065,A -85,B 0,C 180,E1 -22081.532,E2 -22081.532} C_VEL
LIN {X 0,Y 198.269,Z 257.015,A -85,B 0,C 180,E1 -22083.667,E2 -22083.667} C_VEL
LIN {X 0,Y 197.045,Z 246.022,A -85,B 0,C 180,E1 -22085.778,E2 -22085.778} C_VEL
LIN {X 0,Y 194.695,Z 234.405,A -85,B 0,C 180,E1 -22087.853,E2 -22087.853} C_VEL
LIN {X 0,Y 191.993,Z 226.178,A -85,B 0,C 180,E1 -22089.349,E2 -22089.349} C_VEL
LIN {X 0,Y 189.434,Z 220.136,A -85,B 0,C 180,E1 -22090.504,E2 -22090.504} C_VEL
LIN {X 0,Y 187.728,Z 216.846,A -85,B 0,C 180,E1 -22091.197,E2 -22091.197} C_VEL
LIN {X 0,Y 187.453,Z 215.595,A -85,B 0,C 180,E1 -22091.423,E2 -22091.423} C_VEL
LIN {X 0,Y 186.915,Z 212.726,A -85,B 0,C 180,E1 -22095.593,E2 -22095.593} C_VEL
LIN {X 0,Y 186.411,Z 209.812,A -85,B 0,C 180,E1 -22100.139,E2 -22100.139} C_VEL
LIN {X 0,Y 185.942,Z 206.688,A -85,B 0,C 180,E1 -22105.462,E2 -22105.462} C_VEL
LIN {X 0,Y 185.566,Z 204.396,A -85,B 0,C 180,E1 -22109.879,E2 -22109.879} C_VEL
LIN {X 0,Y 185.579,Z 204.372,A -85,B 0,C 180,E1 -22115.381,E2 -22115.381} C_VEL
LIN {X 0,Y 185.673,Z 204.359,A -85,B 0,C 180,E1 -22121.133,E2 -22121.133} C_VEL
LIN {X 0,Y 185.694,Z 204.355,A -85,B 0,C 180,E1 -22124.637,E2 -22124.637} C_VEL
LIN {X 0,Y 185.886,Z 204.322,A -85,B 0,C 180,E1 -22129.419,E2 -22129.419} C_VEL
LIN {X 0,Y 185.934,Z 204.324,A -85,B 0,C 180,E1 -22133.489,E2 -22133.489} C_VEL
LIN {X 0,Y 186.201,Z 204.289,A -85,B 0,C 180,E1 -22137.837,E2 -22137.837} C_VEL
LIN {X 0,Y 186.405,Z 204.266,A -85,B 0,C 180,E1 -22140,E2 -22140} C_VEL
LIN {X 0,Y 185.907,Z 204.325,A -85,B 0,C 180,E1 -22144.336,E2 -22144.336} C_VEL
LIN {X 0,Y 185.974,Z 204.32,A -85,B 0,C 180,E1 -22148.694,E2 -22148.694} C_VEL
LIN {X 0,Y 185.728,Z 204.348,A -85,B 0,C 180,E1 -22153.123,E2 -22153.123} C_VEL
LIN {X 0,Y 185.689,Z 204.355,A -85,B 0,C 180,E1 -22157.625,E2 -22157.625} C_VEL
LIN {X 0,Y 185.596,Z 204.367,A -85,B 0,C 180,E1 -22162.252,E2 -22162.252} C_VEL
LIN {X 0,Y 185.562,Z 204.371,A -85,B 0,C 180,E1 -22167.032,E2 -22167.032} C_VEL
LIN {X 0,Y 185.577,Z 204.368,A -85,B 0,C 180,E1 -22169.494,E2 -22169.494} C_VEL
LIN {X 0,Y 185.497,Z 204.38,A -85,B 0,C 180,E1 -22174.633,E2 -22174.633} C_VEL
LIN {X 0,Y 185.502,Z 204.376,A -85,B 0,C 180,E1 -22177.314,E2 -22177.314} C_VEL
LIN {X 0,Y 185.468,Z 204.385,A -85,B 0,C 180,E1 -22180.725,E2 -22180.725} C_VEL
LIN {X 0,Y 185.669,Z 205.568,A -85,B 0,C 180,E1 -22184.013,E2 -22184.013} C_VEL
LIN {X 0,Y 185.961,Z 207.724,A -85,B 0,C 180,E1 -22188.32,E2 -22188.32} C_VEL
LIN {X 0,Y 187.14,Z 210.759,A -85,B 0,C 180,E1 -22188.879,E2 -22188.879} C_VEL
LIN {X 0,Y 188.626,Z 213.065,A -85,B 0,C 180,E1 -22189.455,E2 -22189.455} C_VEL
LIN {X 0,Y 192.676,Z 221.81,A -85,B 0,C 180,E1 -22191.336,E2 -22191.336} C_VEL
LIN {X 0,Y 195.843,Z 230.502,A -85,B 0,C 180,E1 -22193.14,E2 -22193.14} C_VEL
LIN {X 0,Y 198.305,Z 240.214,A -85,B 0,C 180,E1 -22195.141,E2 -22195.141} C_VEL
LIN {X 0,Y 199.855,Z 249.404,A -85,B 0,C 180,E1 -22197.136,E2 -22197.136} C_VEL
LIN {X 0,Y 200.703,Z 259.437,A -85,B 0,C 180,E1 -22199.487,E2 -22199.487} C_VEL
LIN {X 0,Y 200.561,Z 262.926,A -85,B 0,C 180,E1 -22200.333,E2 -22200.333} C_VEL
LIN {X 0,Y 197.682,Z 272.231,A -85,B 0,C 180,E1 -22202.473,E2 -22202.473} C_VEL
LIN {X 0,Y 194.943,Z 280.699,A -85,B 0,C 180,E1 -22204.938,E2 -22204.938} C_VEL
LIN {X 0,Y 191.848,Z 288.939,A -85,B 0,C 180,E1 -22207.946,E2 -22207.946} C_VEL
LIN {X 0,Y 189.562,Z 294.576,A -85,B 0,C 180,E1 -22210.509,E2 -22210.509} C_VEL
LIN {X 0,Y 187.412,Z 300.064,A -85,B 0,C 180,E1 -22213.666,E2 -22213.666} C_VEL
LIN {X 0,Y 185.671,Z 304.371,A -85,B 0,C 180,E1 -22216.874,E2 -22216.874} C_VEL
LIN {X 0,Y 184.855,Z 306.647,A -85,B 0,C 180,E1 -22219.042,E2 -22219.042} C_VEL
LIN {X 0,Y 184.178,Z 308.497,A -85,B 0,C 180,E1 -22221.221,E2 -22221.221} C_VEL
LIN {X 0,Y 183.53,Z 310.509,A -85,B 0,C 180,E1 -22224.644,E2 -22224.644} C_VEL
LIN {X 0,Y 183.251,Z 311.479,A -85,B 0,C 180,E1 -22227.803,E2 -22227.803} C_VEL
LIN {X 0,Y 183.234,Z 311.704,A -85,B 0,C 180,E1 -22230.001,E2 -22230.001} C_VEL
LIN {X 0,Y 183.25,Z 311.51,A -85,B 0,C 180,E1 -22232.198,E2 -22232.198} C_VEL
LIN {X 0,Y 183.738,Z 309.956,A -85,B 0,C 180,E1 -22236.59,E2 -22236.59} C_VEL
LIN {X 0,Y 184.176,Z 308.6,A -85,B 0,C 180,E1 -22238.78,E2 -22238.78} C_VEL
LIN {X 0,Y 185.217,Z 305.733,A -85,B 0,C 180,E1 -22242.046,E2 -22242.046} C_VEL
LIN {X 0,Y 186.735,Z 301.841,A -85,B 0,C 180,E1 -22245.276,E2 -22245.276} C_VEL
LIN {X 0,Y 188.751,Z 296.82,A -85,B 0,C 180,E1 -22248.451,E2 -22248.451} C_VEL
LIN {X 0,Y 191.299,Z 290.49,A -85,B 0,C 180,E1 -22251.555,E2 -22251.555} C_VEL
LIN {X 0,Y 194.399,Z 282.569,A -85,B 0,C 180,E1 -22254.567,E2 -22254.567} C_VEL
LIN {X 0,Y 197.087,Z 274.369,A -85,B 0,C 180,E1 -22257.086,E2 -22257.086} C_VEL
LIN {X 0,Y 200.147,Z 264.648,A -85,B 0,C 180,E1 -22259.446,E2 -22259.446} C_VEL
LIN {X 0,Y 200.76,Z 262.377,A -85,B 0,C 180,E1 -22259.924,E2 -22259.924} C_VEL
LIN {X 0,Y 200.235,Z 252.541,A -85,B 0,C 180,E1 -22262.298,E2 -22262.298} C_VEL
LIN {X 0,Y 198.847,Z 242.902,A -85,B 0,C 180,E1 -22264.438,E2 -22264.438} C_VEL
LIN {X 0,Y 196.651,Z 233.175,A -85,B 0,C 180,E1 -22266.466,E2 -22266.466} C_VEL
LIN {X 0,Y 193.133,Z 222.724,A -85,B 0,C 180,E1 -22268.624,E2 -22268.624} C_VEL
LIN {X 0,Y 189.74,Z 215.413,A -85,B 0,C 180,E1 -22270.22,E2 -22270.22} C_VEL
LIN {X 0,Y 187.907,Z 211.842,A -85,B 0,C 180,E1 -22271.008,E2 -22271.008} C_VEL
LIN {X 0,Y 186.227,Z 208.843,A -85,B 0,C 180,E1 -22271.703,E2 -22271.703} C_VEL
LIN {X 0,Y 185.921,Z 207.691,A -85,B 0,C 180,E1 -22271.878,E2 -22271.878} C_VEL
LIN {X 0,Y 185.601,Z 205.147,A -85,B 0,C 180,E1 -22277.031,E2 -22277.031} C_VEL
LIN {X 0,Y 185.468,Z 204.384,A -85,B 0,C 180,E1 -22279.895,E2 -22279.895} C_VEL
LIN {X 0,Y 185.506,Z 204.377,A -85,B 0,C 180,E1 -22282.712,E2 -22282.712} C_VEL
LIN {X 0,Y 185.544,Z 204.37,A -85,B 0,C 180,E1 -22287.975,E2 -22287.975} C_VEL
LIN {X 0,Y 185.582,Z 204.365,A -85,B 0,C 180,E1 -22290.577,E2 -22290.577} C_VEL
LIN {X 0,Y 185.59,Z 204.367,A -85,B 0,C 180,E1 -22295.383,E2 -22295.383} C_VEL
LIN {X 0,Y 185.677,Z 204.353,A -85,B 0,C 180,E1 -22301.133,E2 -22301.133} C_VEL
LIN {X 0,Y 185.697,Z 204.354,A -85,B 0,C 180,E1 -22304.637,E2 -22304.637} C_VEL
LIN {X 0,Y 185.89,Z 204.331,A -85,B 0,C 180,E1 -22309.419,E2 -22309.419} C_VEL
LIN {X 0,Y 185.938,Z 204.323,A -85,B 0,C 180,E1 -22313.489,E2 -22313.489} C_VEL
LIN {X 0,Y 186.203,Z 204.289,A -85,B 0,C 180,E1 -22317.837,E2 -22317.837} C_VEL
LIN {X 0,Y 186.408,Z 204.263,A -85,B 0,C 180,E1 -22320,E2 -22320} C_VEL
LIN {X 0,Y 185.91,Z 204.329,A -85,B 0,C 180,E1 -22324.336,E2 -22324.336} C_VEL
LIN {X 0,Y 185.976,Z 204.323,A -85,B 0,C 180,E1 -22328.694,E2 -22328.694} C_VEL
LIN {X 0,Y 185.733,Z 204.353,A -85,B 0,C 180,E1 -22333.123,E2 -22333.123} C_VEL
LIN {X 0,Y 185.692,Z 204.357,A -85,B 0,C 180,E1 -22337.625,E2 -22337.625} C_VEL
LIN {X 0,Y 185.583,Z 204.368,A -85,B 0,C 180,E1 -22342.253,E2 -22342.253} C_VEL
LIN {X 0,Y 185.56,Z 204.373,A -85,B 0,C 180,E1 -22347.032,E2 -22347.032} C_VEL
LIN {X 0,Y 185.571,Z 204.455,A -85,B 0,C 180,E1 -22350.12,E2 -22350.12} C_VEL
LIN {X 0,Y 185.945,Z 206.767,A -85,B 0,C 180,E1 -22354.537,E2 -22354.537} C_VEL
LIN {X 0,Y 186.219,Z 208.486,A -85,B 0,C 180,E1 -22357.575,E2 -22357.575} C_VEL
LIN {X 0,Y 186.697,Z 211.638,A -85,B 0,C 180,E1 -22362.656,E2 -22362.656} C_VEL
LIN {X 0,Y 187.381,Z 215.35,A -85,B 0,C 180,E1 -22368.156,E2 -22368.156} C_VEL
LIN {X 0,Y 187.444,Z 215.735,A -85,B 0,C 180,E1 -22368.58,E2 -22368.58} C_VEL
LIN {X 0,Y 188.491,Z 218.755,A -85,B 0,C 180,E1 -22369.069,E2 -22369.069} C_VEL
LIN {X 0,Y 189.791,Z 220.862,A -85,B 0,C 180,E1 -22369.566,E2 -22369.566} C_VEL
LIN {X 0,Y 193.037,Z 228.991,A -85,B 0,C 180,E1 -22371.098,E2 -22371.098} C_VEL
LIN {X 0,Y 195.165,Z 236.118,A -85,B 0,C 180,E1 -22372.395,E2 -22372.395} C_VEL
LIN {X 0,Y 197.349,Z 247.511,A -85,B 0,C 180,E1 -22374.452,E2 -22374.452} C_VEL
LIN {X 0,Y 198.372,Z 258.525,A -85,B 0,C 180,E1 -22376.58,E2 -22376.58} C_VEL
LIN {X 0,Y 198.572,Z 268.476,A -85,B 0,C 180,E1 -22378.729,E2 -22378.729} C_VEL
LIN {X 0,Y 198.062,Z 278.11,A -85,B 0,C 180,E1 -22381.087,E2 -22381.087} C_VEL
LIN {X 0,Y 195.2,Z 286.63,A -85,B 0,C 180,E1 -22383.253,E2 -22383.253} C_VEL
LIN {X 0,Y 192.419,Z 294.642,A -85,B 0,C 180,E1 -22385.796,E2 -22385.796} C_VEL
LIN {X 0,Y 189.663,Z 302.184,A -85,B 0,C 180,E1 -22388.82,E2 -22388.82} C_VEL
LIN {X 0,Y 186.955,Z 309.276,A -85,B 0,C 180,E1 -22392.498,E2 -22392.498} C_VEL
LIN {X 0,Y 185.227,Z 313.997,A -85,B 0,C 180,E1 -22395.722,E2 -22395.722} C_VEL
LIN {X 0,Y 183.986,Z 317.896,A -85,B 0,C 180,E1 -22399.331,E2 -22399.331} C_VEL
LIN {X 0,Y 183.551,Z 319.473,A -85,B 0,C 180,E1 -22401.19,E2 -22401.19} C_VEL
LIN {X 0,Y 183.23,Z 320.872,A -85,B 0,C 180,E1 -22403.392,E2 -22403.392} C_VEL
LIN {X 0,Y 183.038,Z 322.232,A -85,B 0,C 180,E1 -22406.666,E2 -22406.666} C_VEL
LIN {X 0,Y 183.079,Z 322.582,A -85,B 0,C 180,E1 -22408.774,E2 -22408.774} C_VEL
LIN {X 0,Y 182.435,Z 322.653,A -85,B 0,C 180,E1 -22410.609,E2 -22410.609} C_VEL
LIN {X 0,Y 180.839,Z 322.39,A -85,B 0,C 180,E1 -22412.413,E2 -22412.413} C_VEL
LIN {X 0,Y 177.204,Z 321.058,A -85,B 0,C 180,E1 -22416.055,E2 -22416.055} C_VEL
LIN {X 0,Y 176.367,Z 320.015,A -85,B 0,C 180,E1 -22417.947,E2 -22417.947} C_VEL
LIN {X 0,Y 176.392,Z 319.584,A -85,B 0,C 180,E1 -22418.584,E2 -22418.584} C_VEL
LIN {X 0,Y 177.449,Z 316.272,A -85,B 0,C 180,E1 -22422.581,E2 -22422.581} C_VEL
LIN {X 0,Y 178.815,Z 312.278,A -85,B 0,C 180,E1 -22425.969,E2 -22425.969} C_VEL
LIN {X 0,Y 181.351,Z 306.151,A -85,B 0,C 180,E1 -22429.821,E2 -22429.821} C_VEL
LIN {X 0,Y 184.021,Z 299.588,A -85,B 0,C 180,E1 -22432.985,E2 -22432.985} C_VEL
LIN {X 0,Y 187.028,Z 291.159,A -85,B 0,C 180,E1 -22436.201,E2 -22436.201} C_VEL
LIN {X 0,Y 190.12,Z 282.654,A -85,B 0,C 180,E1 -22438.721,E2 -22438.721} C_VEL
LIN {X 0,Y 191.445,Z 278.74,A -85,B 0,C 180,E1 -22439.708,E2 -22439.708} C_VEL
LIN {X 0,Y 192.178,Z 268.061,A -85,B 0,C 180,E1 -22442.42,E2 -22442.42} C_VEL
LIN {X 0,Y 191.948,Z 257.689,A -85,B 0,C 180,E1 -22444.752,E2 -22444.752} C_VEL
LIN {X 0,Y 190.833,Z 246.737,A -85,B 0,C 180,E1 -22446.977,E2 -22446.977} C_VEL
LIN {X 0,Y 188.676,Z 235.771,A -85,B 0,C 180,E1 -22449.078,E2 -22449.078} C_VEL
LIN {X 0,Y 185.723,Z 227.346,A -85,B 0,C 180,E1 -22450.815,E2 -22450.815} C_VEL
LIN {X 0,Y 184.253,Z 224.046,A -85,B 0,C 180,E1 -22451.531,E2 -22451.531} C_VEL
LIN {X 0,Y 182.342,Z 220.031,A -85,B 0,C 180,E1 -22452.419,E2 -22452.419} C_VEL
LIN {X 0,Y 180.473,Z 216.663,A -85,B 0,C 180,E1 -22453.235,E2 -22453.235} C_VEL
LIN {X 0,Y 180.146,Z 215.339,A -85,B 0,C 180,E1 -22453.47,E2 -22453.47} C_VEL
LIN {X 0,Y 179.601,Z 212.268,A -85,B 0,C 180,E1 -22458.3,E2 -22458.3} C_VEL
LIN {X 0,Y 179.294,Z 210.286,A -85,B 0,C 180,E1 -22461.624,E2 -22461.624} C_VEL
LIN {X 0,Y 178.917,Z 207.524,A -85,B 0,C 180,E1 -22466.638,E2 -22466.638} C_VEL
LIN {X 0,Y 178.509,Z 205.251,A -85,B 0,C 180,E1 -22471.572,E2 -22471.572} C_VEL
LIN {X 0,Y 178.497,Z 205.254,A -85,B 0,C 180,E1 -22476.813,E2 -22476.813} C_VEL
LIN {X 0,Y 178.648,Z 205.233,A -85,B 0,C 180,E1 -22481.656,E2 -22481.656} C_VEL
LIN {X 0,Y 178.656,Z 205.231,A -85,B 0,C 180,E1 -22486.348,E2 -22486.348} C_VEL
LIN {X 0,Y 178.903,Z 205.198,A -85,B 0,C 180,E1 -22490.959,E2 -22490.959} C_VEL
LIN {X 0,Y 179.146,Z 205.168,A -85,B 0,C 180,E1 -22497.752,E2 -22497.752} C_VEL
LIN {X 0,Y 179.368,Z 205.142,A -85,B 0,C 180,E1 -22500,E2 -22500} C_VEL
LIN {X 0,Y 178.855,Z 205.204,A -85,B 0,C 180,E1 -22504.508,E2 -22504.508} C_VEL
LIN {X 0,Y 178.904,Z 205.199,A -85,B 0,C 180,E1 -22509.041,E2 -22509.041} C_VEL
LIN {X 0,Y 178.656,Z 205.23,A -85,B 0,C 180,E1 -22513.652,E2 -22513.652} C_VEL
LIN {X 0,Y 178.622,Z 205.235,A -85,B 0,C 180,E1 -22519.217,E2 -22519.217} C_VEL
LIN {X 0,Y 178.534,Z 205.246,A -85,B 0,C 180,E1 -22525.125,E2 -22525.125} C_VEL
LIN {X 0,Y 178.521,Z 205.248,A -85,B 0,C 180,E1 -22529.994,E2 -22529.994} C_VEL
LIN {X 0,Y 178.483,Z 205.254,A -85,B 0,C 180,E1 -22534.219,E2 -22534.219} C_VEL
LIN {X 0,Y 178.393,Z 205.266,A -85,B 0,C 180,E1 -22539.076,E2 -22539.076} C_VEL
LIN {X 0,Y 178.546,Z 206.033,A -85,B 0,C 180,E1 -22542.003,E2 -22542.003} C_VEL
LIN {X 0,Y 178.864,Z 208.03,A -85,B 0,C 180,E1 -22546.271,E2 -22546.271} C_VEL
LIN {X 0,Y 180.003,Z 210.974,A -85,B 0,C 180,E1 -22546.856,E2 -22546.856} C_VEL
LIN {X 0,Y 181.839,Z 213.849,A -85,B 0,C 180,E1 -22547.641,E2 -22547.641} C_VEL
LIN {X 0,Y 185.698,Z 221.432,A -85,B 0,C 180,E1 -22549.514,E2 -22549.514} C_VEL
LIN {X 0,Y 189.563,Z 231.56,A -85,B 0,C 180,E1 -22551.825,E2 -22551.825} C_VEL
LIN {X 0,Y 192.011,Z 241.183,A -85,B 0,C 180,E1 -22553.955,E2 -22553.955} C_VEL
LIN {X 0,Y 193.62,Z 251.32,A -85,B 0,C 180,E1 -22556.297,E2 -22556.297} C_VEL
LIN {X 0,Y 194.28,Z 260.985,A -85,B 0,C 180,E1 -22558.707,E2 -22558.707} C_VEL
LIN {X 0,Y 194.069,Z 264.295,A -85,B 0,C 180,E1 -22559.537,E2 -22559.537} C_VEL
LIN {X 0,Y 191.398,Z 272.448,A -85,B 0,C 180,E1 -22561.488,E2 -22561.488} C_VEL
LIN {X 0,Y 188.528,Z 280.915,A -85,B 0,C 180,E1 -22564.023,E2 -22564.023} C_VEL
LIN {X 0,Y 185.286,Z 289.154,A -85,B 0,C 180,E1 -22567.122,E2 -22567.122} C_VEL
LIN {X 0,Y 182.88,Z 294.791,A -85,B 0,C 180,E1 -22569.766,E2 -22569.766} C_VEL
LIN {X 0,Y 180.594,Z 300.279,A -85,B 0,C 180,E1 -22573.031,E2 -22573.031} C_VEL
LIN {X 0,Y 178.756,Z 304.586,A -85,B 0,C 180,E1 -22576.356,E2 -22576.356} C_VEL
LIN {X 0,Y 177.876,Z 306.862,A -85,B 0,C 180,E1 -22578.607,E2 -22578.607} C_VEL
LIN {X 0,Y 177.174,Z 308.711,A -85,B 0,C 180,E1 -22580.871,E2 -22580.871} C_VEL
LIN {X 0,Y 176.395,Z 310.908,A -85,B 0,C 180,E1 -22584.915,E2 -22584.915} C_VEL
LIN {X 0,Y 176.165,Z 311.692,A -85,B 0,C 180,E1 -22587.714,E2 -22587.714} C_VEL
LIN {X 0,Y 176.142,Z 311.917,A -85,B 0,C 180,E1 -22590.001,E2 -22590.001} C_VEL
LIN {X 0,Y 176.164,Z 311.723,A -85,B 0,C 180,E1 -22592.287,E2 -22592.287} C_VEL
LIN {X 0,Y 176.703,Z 310.168,A -85,B 0,C 180,E1 -22596.853,E2 -22596.853} C_VEL
LIN {X 0,Y 177.172,Z 308.812,A -85,B 0,C 180,E1 -22599.13,E2 -22599.13} C_VEL
LIN {X 0,Y 178.261,Z 305.945,A -85,B 0,C 180,E1 -22602.524,E2 -22602.524} C_VEL
LIN {X 0,Y 179.875,Z 302.054,A -85,B 0,C 180,E1 -22605.873,E2 -22605.873} C_VEL
LIN {X 0,Y 182.032,Z 297.031,A -85,B 0,C 180,E1 -22609.158,E2 -22609.158} C_VEL
LIN {X 0,Y 184.714,Z 290.701,A -85,B 0,C 180,E1 -22612.364,E2 -22612.364} C_VEL
LIN {X 0,Y 187.96,Z 282.779,A -85,B 0,C 180,E1 -22615.468,E2 -22615.468} C_VEL
LIN {X 0,Y 190.693,Z 274.818,A -85,B 0,C 180,E1 -22617.993,E2 -22617.993} C_VEL
LIN {X 0,Y 193.985,Z 264.857,A -85,B 0,C 180,E1 -22620.479,E2 -22620.479} C_VEL
LIN {X 0,Y 194.31,Z 262.623,A -85,B 0,C 180,E1 -22621.018,E2 -22621.018} C_VEL
LIN {X 0,Y 193.821,Z 252.834,A -85,B 0,C 180,E1 -22623.489,E2 -22623.489} C_VEL
LIN {X 0,Y 192.429,Z 243.131,A -85,B 0,C 180,E1 -22625.758,E2 -22625.758} C_VEL
LIN {X 0,Y 190.242,Z 233.723,A -85,B 0,C 180,E1 -22627.858,E2 -22627.858} C_VEL
LIN {X 0,Y 187.387,Z 225.393,A -85,B 0,C 180,E1 -22629.747,E2 -22629.747} C_VEL
LIN {X 0,Y 183.421,Z 216.765,A -85,B 0,C 180,E1 -22631.798,E2 -22631.798} C_VEL
LIN {X 0,Y 180.967,Z 212.317,A -85,B 0,C 180,E1 -22632.929,E2 -22632.929} C_VEL
LIN {X 0,Y 179.117,Z 209.109,A -85,B 0,C 180,E1 -22633.763,E2 -22633.763} C_VEL
LIN {X 0,Y 178.845,Z 207.964,A -85,B 0,C 180,E1 -22633.977,E2 -22633.977} C_VEL
LIN {X 0,Y 178.527,Z 205.945,A -85,B 0,C 180,E1 -22638.415,E2 -22638.415} C_VEL
LIN {X 0,Y 178.436,Z 205.26,A -85,B 0,C 180,E1 -22641.975,E2 -22641.975} C_VEL
LIN {X 0,Y 178.487,Z 205.253,A -85,B 0,C 180,E1 -22646.547,E2 -22646.547} C_VEL
LIN {X 0,Y 178.523,Z 205.245,A -85,B 0,C 180,E1 -22650.007,E2 -22650.007} C_VEL
LIN {X 0,Y 178.537,Z 205.243,A -85,B 0,C 180,E1 -22654.876,E2 -22654.876} C_VEL
LIN {X 0,Y 178.625,Z 205.233,A -85,B 0,C 180,E1 -22660.784,E2 -22660.784} C_VEL
LIN {X 0,Y 178.66,Z 205.231,A -85,B 0,C 180,E1 -22666.348,E2 -22666.348} C_VEL
LIN {X 0,Y 178.908,Z 205.198,A -85,B 0,C 180,E1 -22670.959,E2 -22670.959} C_VEL
LIN {X 0,Y 179.149,Z 205.168,A -85,B 0,C 180,E1 -22677.752,E2 -22677.752} C_VEL
LIN {X 0,Y 179.371,Z 205.14,A -85,B 0,C 180,E1 -22680,E2 -22680} C_VEL
LIN {X 0,Y 178.857,Z 205.208,A -85,B 0,C 180,E1 -22684.507,E2 -22684.507} C_VEL
LIN {X 0,Y 178.906,Z 205.202,A -85,B 0,C 180,E1 -22689.04,E2 -22689.04} C_VEL
LIN {X 0,Y 178.661,Z 205.233,A -85,B 0,C 180,E1 -22693.652,E2 -22693.652} C_VEL
LIN {X 0,Y 178.624,Z 205.237,A -85,B 0,C 180,E1 -22699.215,E2 -22699.215} C_VEL
LIN {X 0,Y 178.521,Z 205.249,A -85,B 0,C 180,E1 -22705.114,E2 -22705.114} C_VEL
LIN {X 0,Y 178.487,Z 205.255,A -85,B 0,C 180,E1 -22708.197,E2 -22708.197} C_VEL
LIN {X 0,Y 178.684,Z 206.294,A -85,B 0,C 180,E1 -22710.752,E2 -22710.752} C_VEL
LIN {X 0,Y 179.003,Z 208.173,A -85,B 0,C 180,E1 -22714.462,E2 -22714.462} C_VEL
LIN {X 0,Y 179.349,Z 210.603,A -85,B 0,C 180,E1 -22718.828,E2 -22718.828} C_VEL
LIN {X 0,Y 179.965,Z 214.173,A -85,B 0,C 180,E1 -22724.663,E2 -22724.663} C_VEL
LIN {X 0,Y 180.186,Z 215.564,A -85,B 0,C 180,E1 -22726.516,E2 -22726.516} C_VEL
LIN {X 0,Y 181.435,Z 218.755,A -85,B 0,C 180,E1 -22727.13,E2 -22727.13} C_VEL
LIN {X 0,Y 182.911,Z 221.094,A -85,B 0,C 180,E1 -22727.743,E2 -22727.743} C_VEL
LIN {X 0,Y 186.644,Z 229.497,A -85,B 0,C 180,E1 -22729.582,E2 -22729.582} C_VEL
LIN {X 0,Y 189.224,Z 237.909,A -85,B 0,C 180,E1 -22731.258,E2 -22731.258} C_VEL
LIN {X 0,Y 191.334,Z 249.87,A -85,B 0,C 180,E1 -22733.581,E2 -22733.581} C_VEL
LIN {X 0,Y 192.15,Z 261.399,A -85,B 0,C 180,E1 -22735.993,E2 -22735.993} C_VEL
LIN {X 0,Y 192.111,Z 270.505,A -85,B 0,C 180,E1 -22738.108,E2 -22738.108} C_VEL
LIN {X 0,Y 191.504,Z 278.936,A -85,B 0,C 180,E1 -22740.301,E2 -22740.301} C_VEL
LIN {X 0,Y 188.257,Z 288.091,A -85,B 0,C 180,E1 -22742.785,E2 -22742.785} C_VEL
LIN {X 0,Y 185.299,Z 296.121,A -85,B 0,C 180,E1 -22745.543,E2 -22745.543} C_VEL
LIN {X 0,Y 182.562,Z 303.093,A -85,B 0,C 180,E1 -22748.548,E2 -22748.548} C_VEL
LIN {X 0,Y 180.167,Z 309.063,A -85,B 0,C 180,E1 -22751.816,E2 -22751.816} C_VEL
LIN {X 0,Y 178.317,Z 313.784,A -85,B 0,C 180,E1 -22755.156,E2 -22755.156} C_VEL
LIN {X 0,Y 177.081,Z 317.396,A -85,B 0,C 180,E1 -22758.554,E2 -22758.554} C_VEL
LIN {X 0,Y 176.509,Z 319.26,A -85,B 0,C 180,E1 -22760.835,E2 -22760.835} C_VEL
LIN {X 0,Y 176.008,Z 321.661,A -85,B 0,C 180,E1 -22765.419,E2 -22765.419} C_VEL
LIN {X 0,Y 175.983,Z 322.376,A -85,B 0,C 180,E1 -22768.806,E2 -22768.806} C_VEL
LIN {X 0,Y 176.071,Z 322.489,A -85,B 0,C 180,E1 -22769.999,E2 -22769.999} C_VEL
LIN {X 0,Y 175.97,Z 322.073,A -85,B 0,C 180,E1 -22773.175,E2 -22773.175} C_VEL
LIN {X 0,Y 176.155,Z 320.636,A -85,B 0,C 180,E1 -22776.874,E2 -22776.874} C_VEL
LIN {X 0,Y 176.392,Z 319.584,A -85,B 0,C 180,E1 -22778.584,E2 -22778.584} C_VEL
LIN {X 0,Y 176.128,Z 318.279,A -85,B 0,C 180,E1 -22780.455,E2 -22780.455} C_VEL
LIN {X 0,Y 174.185,Z 315.545,A -85,B 0,C 180,E1 -22783.511,E2 -22783.511} C_VEL
LIN {X 0,Y 172.648,Z 312.091,A -85,B 0,C 180,E1 -22786.55,E2 -22786.55} C_VEL
LIN {X 0,Y 173.022,Z 309.633,A -85,B 0,C 180,E1 -22788.334,E2 -22788.334} C_VEL
LIN {X 0,Y 175.472,Z 303.891,A -85,B 0,C 180,E1 -22791.745,E2 -22791.745} C_VEL
LIN {X 0,Y 178.143,Z 297.635,A -85,B 0,C 180,E1 -22794.652,E2 -22794.652} C_VEL
LIN {X 0,Y 181.29,Z 289.35,A -85,B 0,C 180,E1 -22797.722,E2 -22797.722} C_VEL
LIN {X 0,Y 184.622,Z 280.485,A -85,B 0,C 180,E1 -22800.29,E2 -22800.29} C_VEL
LIN {X 0,Y 185.6,Z 272.947,A -85,B 0,C 180,E1 -22802.362,E2 -22802.362} C_VEL
LIN {X 0,Y 185.881,Z 264.243,A -85,B 0,C 180,E1 -22804.55,E2 -22804.55} C_VEL
LIN {X 0,Y 185.339,Z 253.201,A -85,B 0,C 180,E1 -22807.047,E2 -22807.047} C_VEL
LIN {X 0,Y 183.684,Z 241.673,A -85,B 0,C 180,E1 -22809.464,E2 -22809.464} C_VEL
LIN {X 0,Y 181.608,Z 233.876,A -85,B 0,C 180,E1 -22811.137,E2 -22811.137} C_VEL
LIN {X 0,Y 178.016,Z 225.079,A -85,B 0,C 180,E1 -22813.197,E2 -22813.197} C_VEL
LIN {X 0,Y 175.944,Z 221.232,A -85,B 0,C 180,E1 -22814.223,E2 -22814.223} C_VEL
LIN {X 0,Y 175.076,Z 219.761,A -85,B 0,C 180,E1 -22814.627,E2 -22814.627} C_VEL
LIN {X 0,Y 173.282,Z 216.498,A -85,B 0,C 180,E1 -22815.501,E2 -22815.501} C_VEL
LIN {X 0,Y 172.899,Z 215.061,A -85,B 0,C 180,E1 -22815.784,E2 -22815.784} C_VEL
LIN {X 0,Y 172.371,Z 212.113,A -85,B 0,C 180,E1 -22820.774,E2 -22820.774} C_VEL
LIN {X 0,Y 172.054,Z 209.782,A -85,B 0,C 180,E1 -22825.119,E2 -22825.119} C_VEL
LIN {X 0,Y 171.655,Z 207.153,A -85,B 0,C 180,E1 -22830.573,E2 -22830.573} C_VEL
LIN {X 0,Y 171.412,Z 206.136,A -85,B 0,C 180,E1 -22833.192,E2 -22833.192} C_VEL
LIN {X 0,Y 171.452,Z 206.131,A -85,B 0,C 180,E1 -22838.351,E2 -22838.351} C_VEL
LIN {X 0,Y 171.577,Z 206.115,A -85,B 0,C 180,E1 -22840.871,E2 -22840.871} C_VEL
LIN {X 0,Y 171.574,Z 206.112,A -85,B 0,C 180,E1 -22845.773,E2 -22845.773} C_VEL
LIN {X 0,Y 171.841,Z 206.076,A -85,B 0,C 180,E1 -22850.585,E2 -22850.585} C_VEL
LIN {X 0,Y 171.802,Z 206.083,A -85,B 0,C 180,E1 -22855.307,E2 -22855.307} C_VEL
LIN {X 0,Y 172.331,Z 206.019,A -85,B 0,C 180,E1 -22860,E2 -22860} C_VEL
LIN {X 0,Y 171.803,Z 206.083,A -85,B 0,C 180,E1 -22864.693,E2 -22864.693} C_VEL
LIN {X 0,Y 171.842,Z 206.078,A -85,B 0,C 180,E1 -22869.416,E2 -22869.416} C_VEL
LIN {X 0,Y 171.575,Z 206.114,A -85,B 0,C 180,E1 -22874.228,E2 -22874.228} C_VEL
LIN {X 0,Y 171.544,Z 206.117,A -85,B 0,C 180,E1 -22879.563,E2 -22879.563} C_VEL
LIN {X 0,Y 171.468,Z 206.125,A -85,B 0,C 180,E1 -22885.617,E2 -22885.617} C_VEL
LIN {X 0,Y 171.44,Z 206.13,A -85,B 0,C 180,E1 -22890.587,E2 -22890.587} C_VEL
LIN {X 0,Y 171.391,Z 206.137,A -85,B 0,C 180,E1 -22895.035,E2 -22895.035} C_VEL
LIN {X 0,Y 171.355,Z 206.151,A -85,B 0,C 180,E1 -22898.807,E2 -22898.807} C_VEL
LIN {X 0,Y 171.672,Z 208.328,A -85,B 0,C 180,E1 -22903.926,E2 -22903.926} C_VEL
LIN {X 0,Y 172.808,Z 211.172,A -85,B 0,C 180,E1 -22904.566,E2 -22904.566} C_VEL
LIN {X 0,Y 174.639,Z 213.622,A -85,B 0,C 180,E1 -22905.399,E2 -22905.399} C_VEL
LIN {X 0,Y 176.796,Z 217.608,A -85,B 0,C 180,E1 -22906.509,E2 -22906.509} C_VEL
LIN {X 0,Y 180.59,Z 225.358,A -85,B 0,C 180,E1 -22908.58,E2 -22908.58} C_VEL
LIN {X 0,Y 184.068,Z 235.155,A -85,B 0,C 180,E1 -22911.001,E2 -22911.001} C_VEL
LIN {X 0,Y 186.239,Z 244.804,A -85,B 0,C 180,E1 -22913.311,E2 -22913.311} C_VEL
LIN {X 0,Y 187.551,Z 254.782,A -85,B 0,C 180,E1 -22915.801,E2 -22915.801} C_VEL
LIN {X 0,Y 187.908,Z 262.565,A -85,B 0,C 180,E1 -22917.889,E2 -22917.889} C_VEL
LIN {X 0,Y 187.608,Z 265.583,A -85,B 0,C 180,E1 -22918.684,E2 -22918.684} C_VEL
LIN {X 0,Y 184.173,Z 275.563,A -85,B 0,C 180,E1 -22921.274,E2 -22921.274} C_VEL
LIN {X 0,Y 181.054,Z 284.085,A -85,B 0,C 180,E1 -22924.108,E2 -22924.108} C_VEL
LIN {X 0,Y 177.702,Z 291.761,A -85,B 0,C 180,E1 -22927.319,E2 -22927.319} C_VEL
LIN {X 0,Y 174.574,Z 298.805,A -85,B 0,C 180,E1 -22931.213,E2 -22931.213} C_VEL
LIN {X 0,Y 172.451,Z 303.493,A -85,B 0,C 180,E1 -22934.64,E2 -22934.64} C_VEL
LIN {X 0,Y 170.923,Z 307.076,A -85,B 0,C 180,E1 -22938.137,E2 -22938.137} C_VEL
LIN {X 0,Y 170.161,Z 308.925,A -85,B 0,C 180,E1 -22940.491,E2 -22940.491} C_VEL
LIN {X 0,Y 169.66,Z 310.311,A -85,B 0,C 180,E1 -22942.862,E2 -22942.862} C_VEL
LIN {X 0,Y 169.081,Z 311.905,A -85,B 0,C 180,E1 -22947.618,E2 -22947.618} C_VEL
LIN {X 0,Y 169.053,Z 312.13,A -85,B 0,C 180,E1 -22950.001,E2 -22950.001} C_VEL
LIN {X 0,Y 169.081,Z 311.935,A -85,B 0,C 180,E1 -22952.383,E2 -22952.383} C_VEL
LIN {X 0,Y 169.66,Z 310.381,A -85,B 0,C 180,E1 -22957.139,E2 -22957.139} C_VEL
LIN {X 0,Y 170.159,Z 309.025,A -85,B 0,C 180,E1 -22959.51,E2 -22959.51} C_VEL
LIN {X 0,Y 171.33,Z 306.158,A -85,B 0,C 180,E1 -22963.039,E2 -22963.039} C_VEL
LIN {X 0,Y 173.04,Z 302.266,A -85,B 0,C 180,E1 -22966.518,E2 -22966.518} C_VEL
LIN {X 0,Y 175.321,Z 297.243,A -85,B 0,C 180,E1 -22969.922,E2 -22969.922} C_VEL
LIN {X 0,Y 178.168,Z 290.912,A -85,B 0,C 180,E1 -22973.233,E2 -22973.233} C_VEL
LIN {X 0,Y 181.572,Z 282.99,A -85,B 0,C 180,E1 -22976.432,E2 -22976.432} C_VEL
LIN {X 0,Y 184.564,Z 274.678,A -85,B 0,C 180,E1 -22979.132,E2 -22979.132} C_VEL
LIN {X 0,Y 187.901,Z 265.067,A -85,B 0,C 180,E1 -22981.577,E2 -22981.577} C_VEL
LIN {X 0,Y 187.659,Z 255.473,A -85,B 0,C 180,E1 -22984.178,E2 -22984.178} C_VEL
LIN {X 0,Y 186.37,Z 245.251,A -85,B 0,C 180,E1 -22986.743,E2 -22986.743} C_VEL
LIN {X 0,Y 184.058,Z 235.013,A -85,B 0,C 180,E1 -22989.203,E2 -22989.203} C_VEL
LIN {X 0,Y 181.053,Z 226.622,A -85,B 0,C 180,E1 -22991.292,E2 -22991.292} C_VEL
LIN {X 0,Y 177.956,Z 220.012,A -85,B 0,C 180,E1 -22993.061,E2 -22993.061} C_VEL
LIN {X 0,Y 176.272,Z 216.842,A -85,B 0,C 180,E1 -22993.932,E2 -22993.932} C_VEL
LIN {X 0,Y 174.105,Z 212.889,A -85,B 0,C 180,E1 -22995.04,E2 -22995.04} C_VEL
LIN {X 0,Y 172.185,Z 209.984,A -85,B 0,C 180,E1 -22995.959,E2 -22995.959} C_VEL
LIN {X 0,Y 171.657,Z 208.253,A -85,B 0,C 180,E1 -22996.366,E2 -22996.366} C_VEL
LIN {X 0,Y 171.389,Z 206.244,A -85,B 0,C 180,E1 -23001.18,E2 -23001.18} C_VEL
LIN {X 0,Y 171.4,Z 206.132,A -85,B 0,C 180,E1 -23005.093,E2 -23005.093} C_VEL
LIN {X 0,Y 171.45,Z 206.125,A -85,B 0,C 180,E1 -23010.534,E2 -23010.534} C_VEL
LIN {X 0,Y 171.46,Z 206.128,A -85,B 0,C 180,E1 -23015.802,E2 -23015.802} C_VEL
LIN {X 0,Y 171.582,Z 206.11,A -85,B 0,C 180,E1 -23020.872,E2 -23020.872} C_VEL
LIN {X 0,Y 171.578,Z 206.112,A -85,B 0,C 180,E1 -23025.773,E2 -23025.773} C_VEL
LIN {X 0,Y 171.846,Z 206.077,A -85,B 0,C 180,E1 -23030.585,E2 -23030.585} C_VEL
LIN {X 0,Y 171.805,Z 206.083,A -85,B 0,C 180,E1 -23035.307,E2 -23035.307} C_VEL
LIN {X 0,Y 172.334,Z 206.017,A -85,B 0,C 180,E1 -23040,E2 -23040} C_VEL
LIN {X 0,Y 171.806,Z 206.085,A -85,B 0,C 180,E1 -23044.693,E2 -23044.693} C_VEL
LIN {X 0,Y 171.845,Z 206.08,A -85,B 0,C 180,E1 -23049.415,E2 -23049.415} C_VEL
LIN {X 0,Y 171.579,Z 206.114,A -85,B 0,C 180,E1 -23054.227,E2 -23054.227} C_VEL
LIN {X 0,Y 171.544,Z 206.119,A -85,B 0,C 180,E1 -23059.559,E2 -23059.559} C_VEL
LIN {X 0,Y 171.46,Z 206.127,A -85,B 0,C 180,E1 -23065.609,E2 -23065.609} C_VEL
LIN {X 0,Y 171.415,Z 206.135,A -85,B 0,C 180,E1 -23066.808,E2 -23066.808} C_VEL
LIN {X 0,Y 171.768,Z 207.824,A -85,B 0,C 180,E1 -23070.769,E2 -23070.769} C_VEL
LIN {X 0,Y 172.071,Z 210.024,A -85,B 0,C 180,E1 -23075.226,E2 -23075.226} C_VEL
LIN {X 0,Y 172.499,Z 213.014,A -85,B 0,C 180,E1 -23080.683,E2 -23080.683} C_VEL
LIN {X 0,Y 172.878,Z 215.06,A -85,B 0,C 180,E1 -23084.122,E2 -23084.122} C_VEL
LIN {X 0,Y 174.238,Z 218.572,A -85,B 0,C 180,E1 -23084.9,E2 -23084.9} C_VEL
LIN {X 0,Y 175.827,Z 220.948,A -85,B 0,C 180,E1 -23085.62,E2 -23085.62} C_VEL
LIN {X 0,Y 177.836,Z 224.862,A -85,B 0,C 180,E1 -23086.635,E2 -23086.635} C_VEL
LIN {X 0,Y 181.464,Z 233.332,A -85,B 0,C 180,E1 -23088.665,E2 -23088.665} C_VEL
LIN {X 0,Y 183.807,Z 242.038,A -85,B 0,C 180,E1 -23090.545,E2 -23090.545} C_VEL
LIN {X 0,Y 185.444,Z 253.353,A -85,B 0,C 180,E1 -23092.933,E2 -23092.933} C_VEL
LIN {X 0,Y 185.901,Z 264.528,A -85,B 0,C 180,E1 -23095.453,E2 -23095.453} C_VEL
LIN {X 0,Y 185.583,Z 273.172,A -85,B 0,C 180,E1 -23097.63,E2 -23097.63} C_VEL
LIN {X 0,Y 185.076,Z 278.716,A -85,B 0,C 180,E1 -23099.16,E2 -23099.16} C_VEL
LIN {X 0,Y 183.955,Z 282.627,A -85,B 0,C 180,E1 -23100.22,E2 -23100.22} C_VEL
LIN {X 0,Y 180.682,Z 291.092,A -85,B 0,C 180,E1 -23102.803,E2 -23102.803} C_VEL
LIN {X 0,Y 177.575,Z 299.178,A -85,B 0,C 180,E1 -23105.971,E2 -23105.971} C_VEL
LIN {X 0,Y 174.663,Z 306.035,A -85,B 0,C 180,E1 -23109.385,E2 -23109.385} C_VEL
LIN {X 0,Y 171.969,Z 312.134,A -85,B 0,C 180,E1 -23113.376,E2 -23113.376} C_VEL
LIN {X 0,Y 170.495,Z 316.108,A -85,B 0,C 180,E1 -23116.896,E2 -23116.896} C_VEL
LIN {X 0,Y 169.487,Z 319.047,A -85,B 0,C 180,E1 -23120.452,E2 -23120.452} C_VEL
LIN {X 0,Y 169.106,Z 320.446,A -85,B 0,C 180,E1 -23122.837,E2 -23122.837} C_VEL
LIN {X 0,Y 168.857,Z 321.999,A -85,B 0,C 180,E1 -23127.32,E2 -23127.32} C_VEL
LIN {X 0,Y 168.98,Z 322.277,A -85,B 0,C 180,E1 -23129.999,E2 -23129.999} C_VEL
LIN {X 0,Y 168.892,Z 321.939,A -85,B 0,C 180,E1 -23132.921,E2 -23132.921} C_VEL
LIN {X 0,Y 169.106,Z 320.422,A -85,B 0,C 180,E1 -23137.162,E2 -23137.162} C_VEL
LIN {X 0,Y 169.487,Z 319.012,A -85,B 0,C 180,E1 -23139.547,E2 -23139.547} C_VEL
LIN {X 0,Y 170.494,Z 316.057,A -85,B 0,C 180,E1 -23143.103,E2 -23143.103} C_VEL
LIN {X 0,Y 171.968,Z 312.063,A -85,B 0,C 180,E1 -23146.623,E2 -23146.623} C_VEL
LIN {X 0,Y 173.022,Z 309.633,A -85,B 0,C 180,E1 -23148.334,E2 -23148.334} C_VEL
LIN {X 0,Y 173.541,Z 307.001,A -85,B 0,C 180,E1 -23150.079,E2 -23150.079} C_VEL
LIN {X 0,Y 172.862,Z 302.337,A -85,B 0,C 180,E1 -23152.976,E2 -23152.976} C_VEL
LIN {X 0,Y 172.424,Z 297.032,A -85,B 0,C 180,E1 -23155.765,E2 -23155.765} C_VEL
LIN {X 0,Y 173.284,Z 293.389,A -85,B 0,C 180,E1 -23157.287,E2 -23157.287} C_VEL
LIN {X 0,Y 177.049,Z 284.025,A -85,B 0,C 180,E1 -23160.405,E2 -23160.405} C_VEL
LIN {X 0,Y 178.381,Z 280.263,A -85,B 0,C 180,E1 -23161.468,E2 -23161.468} C_VEL
LIN {X 0,Y 179.394,Z 271.172,A -85,B 0,C 180,E1 -23164.066,E2 -23164.066} C_VEL
LIN {X 0,Y 179.571,Z 260.817,A -85,B 0,C 180,E1 -23166.717,E2 -23166.717} C_VEL
LIN {X 0,Y 178.765,Z 249.873,A -85,B 0,C 180,E1 -23169.276,E2 -23169.276} C_VEL
LIN {X 0,Y 177.361,Z 241.459,A -85,B 0,C 180,E1 -23171.159,E2 -23171.159} C_VEL
LIN {X 0,Y 174.954,Z 233.596,A -85,B 0,C 180,E1 -23173.07,E2 -23173.07} C_VEL
LIN {X 0,Y 172.628,Z 228.56,A -85,B 0,C 180,E1 -23174.461,E2 -23174.461} C_VEL
LIN {X 0,Y 170.681,Z 224.596,A -85,B 0,C 180,E1 -23175.573,E2 -23175.573} C_VEL
LIN {X 0,Y 168.241,Z 219.944,A -85,B 0,C 180,E1 -23176.925,E2 -23176.925} C_VEL
LIN {X 0,Y 166.2,Z 216.805,A -85,B 0,C 180,E1 -23177.982,E2 -23177.982} C_VEL
LIN {X 0,Y 165.544,Z 214.703,A -85,B 0,C 180,E1 -23178.52,E2 -23178.52} C_VEL
LIN {X 0,Y 165.155,Z 211.796,A -85,B 0,C 180,E1 -23183.951,E2 -23183.951} C_VEL
LIN {X 0,Y 164.855,Z 209.269,A -85,B 0,C 180,E1 -23189.231,E2 -23189.231} C_VEL
LIN {X 0,Y 164.405,Z 207.023,A -85,B 0,C 180,E1 -23194.692,E2 -23194.692} C_VEL
LIN {X 0,Y 164.483,Z 206.998,A -85,B 0,C 180,E1 -23200.051,E2 -23200.051} C_VEL
LIN {X 0,Y 164.522,Z 206.992,A -85,B 0,C 180,E1 -23205.149,E2 -23205.149} C_VEL
LIN {X 0,Y 164.762,Z 206.955,A -85,B 0,C 180,E1 -23210.176,E2 -23210.176} C_VEL
LIN {X 0,Y 164.821,Z 206.953,A -85,B 0,C 180,E1 -23212.651,E2 -23212.651} C_VEL
LIN {X 0,Y 165.041,Z 206.926,A -85,B 0,C 180,E1 -23217.56,E2 -23217.56} C_VEL
LIN {X 0,Y 165.293,Z 206.896,A -85,B 0,C 180,E1 -23220,E2 -23220} C_VEL
LIN {X 0,Y 164.752,Z 206.962,A -85,B 0,C 180,E1 -23224.894,E2 -23224.894} C_VEL
LIN {X 0,Y 164.822,Z 206.952,A -85,B 0,C 180,E1 -23227.35,E2 -23227.35} C_VEL
LIN {X 0,Y 164.701,Z 206.97,A -85,B 0,C 180,E1 -23231.06,E2 -23231.06} C_VEL
LIN {X 0,Y 164.483,Z 206.997,A -85,B 0,C 180,E1 -23237.403,E2 -23237.403} C_VEL
LIN {X 0,Y 164.472,Z 206.998,A -85,B 0,C 180,E1 -23239.989,E2 -23239.989} C_VEL
LIN {X 0,Y 164.393,Z 207.008,A -85,B 0,C 180,E1 -23246.134,E2 -23246.134} C_VEL
LIN {X 0,Y 164.373,Z 207.01,A -85,B 0,C 180,E1 -23251.228,E2 -23251.228} C_VEL
LIN {X 0,Y 164.292,Z 207.018,A -85,B 0,C 180,E1 -23256.79,E2 -23256.79} C_VEL
LIN {X 0,Y 164.535,Z 208.562,A -85,B 0,C 180,E1 -23261.255,E2 -23261.255} C_VEL
LIN {X 0,Y 165.71,Z 211.489,A -85,B 0,C 180,E1 -23262.014,E2 -23262.014} C_VEL
LIN {X 0,Y 167.805,Z 214.356,A -85,B 0,C 180,E1 -23263.09,E2 -23263.09} C_VEL
LIN {X 0,Y 170.021,Z 218.176,A -85,B 0,C 180,E1 -23264.333,E2 -23264.333} C_VEL
LIN {X 0,Y 173.935,Z 225.941,A -85,B 0,C 180,E1 -23266.661,E2 -23266.661} C_VEL
LIN {X 0,Y 177.141,Z 234.011,A -85,B 0,C 180,E1 -23268.922,E2 -23268.922} C_VEL
LIN {X 0,Y 179.451,Z 242.739,A -85,B 0,C 180,E1 -23271.199,E2 -23271.199} C_VEL
LIN {X 0,Y 180.938,Z 252.218,A -85,B 0,C 180,E1 -23273.678,E2 -23273.678} C_VEL
LIN {X 0,Y 181.519,Z 261.324,A -85,B 0,C 180,E1 -23276.19,E2 -23276.19} C_VEL
LIN {X 0,Y 181.498,Z 265.803,A -85,B 0,C 180,E1 -23277.503,E2 -23277.503} C_VEL
LIN {X 0,Y 177.88,Z 276.036,A -85,B 0,C 180,E1 -23280.252,E2 -23280.252} C_VEL
LIN {X 0,Y 174.7,Z 284.301,A -85,B 0,C 180,E1 -23283.092,E2 -23283.092} C_VEL
LIN {X 0,Y 171.18,Z 291.976,A -85,B 0,C 180,E1 -23286.404,E2 -23286.404} C_VEL
LIN {X 0,Y 167.851,Z 299.021,A -85,B 0,C 180,E1 -23290.43,E2 -23290.43} C_VEL
LIN {X 0,Y 165.606,Z 303.708,A -85,B 0,C 180,E1 -23293.988,E2 -23293.988} C_VEL
LIN {X 0,Y 163.99,Z 307.289,A -85,B 0,C 180,E1 -23297.627,E2 -23297.627} C_VEL
LIN {X 0,Y 163.174,Z 309.138,A -85,B 0,C 180,E1 -23300.08,E2 -23300.08} C_VEL
LIN {X 0,Y 162.614,Z 310.525,A -85,B 0,C 180,E1 -23302.551,E2 -23302.551} C_VEL
LIN {X 0,Y 161.988,Z 312.118,A -85,B 0,C 180,E1 -23307.514,E2 -23307.514} C_VEL
LIN {X 0,Y 161.965,Z 312.343,A -85,B 0,C 180,E1 -23310.001,E2 -23310.001} C_VEL
LIN {X 0,Y 162.134,Z 311.729,A -85,B 0,C 180,E1 -23314.449,E2 -23314.449} C_VEL
LIN {X 0,Y 162.614,Z 310.593,A -85,B 0,C 180,E1 -23317.45,E2 -23317.45} C_VEL
LIN {X 0,Y 163.172,Z 309.237,A -85,B 0,C 180,E1 -23319.921,E2 -23319.921} C_VEL
LIN {X 0,Y 164.425,Z 306.37,A -85,B 0,C 180,E1 -23323.597,E2 -23323.597} C_VEL
LIN {X 0,Y 166.238,Z 302.478,A -85,B 0,C 180,E1 -23327.214,E2 -23327.214} C_VEL
LIN {X 0,Y 168.654,Z 297.455,A -85,B 0,C 180,E1 -23330.745,E2 -23330.745} C_VEL
LIN {X 0,Y 171.664,Z 291.123,A -85,B 0,C 180,E1 -23334.168,E2 -23334.168} C_VEL
LIN {X 0,Y 175.238,Z 283.201,A -85,B 0,C 180,E1 -23337.466,E2 -23337.466} C_VEL
LIN {X 0,Y 178.509,Z 274.561,A -85,B 0,C 180,E1 -23340.342,E2 -23340.342} C_VEL
LIN {X 0,Y 181.511,Z 266.342,A -85,B 0,C 180,E1 -23342.496,E2 -23342.496} C_VEL
LIN {X 0,Y 181.436,Z 257.428,A -85,B 0,C 180,E1 -23345.062,E2 -23345.062} C_VEL
LIN {X 0,Y 180.401,Z 247.847,A -85,B 0,C 180,E1 -23347.643,E2 -23347.643} C_VEL
LIN {X 0,Y 178.737,Z 239.35,A -85,B 0,C 180,E1 -23349.844,E2 -23349.844} C_VEL
LIN {X 0,Y 175.786,Z 230.256,A -85,B 0,C 180,E1 -23352.301,E2 -23352.301} C_VEL
LIN {X 0,Y 172.051,Z 222.058,A -85,B 0,C 180,E1 -23354.682,E2 -23354.682} C_VEL
LIN {X 0,Y 169.642,Z 217.691,A -85,B 0,C 180,E1 -23356.062,E2 -23356.062} C_VEL
LIN {X 0,Y 167.699,Z 214.105,A -85,B 0,C 180,E1 -23357.183,E2 -23357.183} C_VEL
LIN {X 0,Y 165.264,Z 210.654,A -85,B 0,C 180,E1 -23358.46,E2 -23358.46} C_VEL
LIN {X 0,Y 164.571,Z 208.563,A -85,B 0,C 180,E1 -23358.959,E2 -23358.959} C_VEL
LIN {X 0,Y 164.295,Z 207.019,A -85,B 0,C 180,E1 -23363.21,E2 -23363.21} C_VEL
LIN {X 0,Y 164.376,Z 207.009,A -85,B 0,C 180,E1 -23368.773,E2 -23368.773} C_VEL
LIN {X 0,Y 164.418,Z 207,A -85,B 0,C 180,E1 -23374.694,E2 -23374.694} C_VEL
LIN {X 0,Y 164.487,Z 206.997,A -85,B 0,C 180,E1 -23380.051,E2 -23380.051} C_VEL
LIN {X 0,Y 164.526,Z 206.99,A -85,B 0,C 180,E1 -23385.149,E2 -23385.149} C_VEL
LIN {X 0,Y 164.767,Z 206.959,A -85,B 0,C 180,E1 -23390.176,E2 -23390.176} C_VEL
LIN {X 0,Y 164.825,Z 206.952,A -85,B 0,C 180,E1 -23392.651,E2 -23392.651} C_VEL
LIN {X 0,Y 165.044,Z 206.925,A -85,B 0,C 180,E1 -23397.559,E2 -23397.559} C_VEL
LIN {X 0,Y 165.296,Z 206.893,A -85,B 0,C 180,E1 -23400,E2 -23400} C_VEL
LIN {X 0,Y 164.754,Z 206.963,A -85,B 0,C 180,E1 -23404.894,E2 -23404.894} C_VEL
LIN {X 0,Y 164.824,Z 206.955,A -85,B 0,C 180,E1 -23407.349,E2 -23407.349} C_VEL
LIN {X 0,Y 164.704,Z 206.972,A -85,B 0,C 180,E1 -23411.059,E2 -23411.059} C_VEL
LIN {X 0,Y 164.485,Z 206.999,A -85,B 0,C 180,E1 -23417.403,E2 -23417.403} C_VEL
LIN {X 0,Y 164.475,Z 206.998,A -85,B 0,C 180,E1 -23419.989,E2 -23419.989} C_VEL
LIN {X 0,Y 164.424,Z 207.081,A -85,B 0,C 180,E1 -23425.305,E2 -23425.305} C_VEL
LIN {X 0,Y 164.845,Z 209.671,A -85,B 0,C 180,E1 -23431.495,E2 -23431.495} C_VEL
LIN {X 0,Y 165.194,Z 212.13,A -85,B 0,C 180,E1 -23436.556,E2 -23436.556} C_VEL
LIN {X 0,Y 165.58,Z 214.77,A -85,B 0,C 180,E1 -23441.479,E2 -23441.479} C_VEL
LIN {X 0,Y 166.751,Z 217.889,A -85,B 0,C 180,E1 -23442.219,E2 -23442.219} C_VEL
LIN {X 0,Y 168.809,Z 220.829,A -85,B 0,C 180,E1 -23443.255,E2 -23443.255} C_VEL
LIN {X 0,Y 170.805,Z 224.774,A -85,B 0,C 180,E1 -23444.386,E2 -23444.386} C_VEL
LIN {X 0,Y 174.054,Z 231.708,A -85,B 0,C 180,E1 -23446.305,E2 -23446.305} C_VEL
